LIN {X -0.095,Y -181.495,Z 926.751,A 0.000,B 0.000,C 90.000,E1 135.162} C_DIS
LIN {X 0.041,Y -187.011,Z 926.732,A 0.000,B 0.000,C 90.000,E1 131.757} C_DIS
LIN {X 0.043,Y -190.129,Z 926.723,A 0.000,B 0.000,C 90.000,E1 130.092} C_DIS
LIN {X -0.054,Y -193.964,Z 926.710,A 0.000,B 0.000,C 90.000,E1 127.890} C_DIS
LIN {X -0.123,Y -295.836,Z 926.710,A 0.000,B 0.000,C 90.000,E1 127.890} C_DIS
LIN {X 0.171,Y -297.593,Z 926.710,A 0.000,B 0.000,C 90.000,E1 127.810} C_DIS
LIN {X -0.111,Y -302.346,Z 926.709,A 0.000,B 0.000,C 90.000,E1 127.649} C_DIS
LIN {X -0.085,Y -305.517,Z 926.707,A 0.000,B 0.000,C 90.000,E1 127.363} C_DIS
LIN {X 0.048,Y -309.189,Z 926.705,A 0.000,B 0.000,C 90.000,E1 126.824} C_DIS
LIN {X 0.011,Y -310.829,Z 926.703,A 0.000,B 0.000,C 90.000,E1 126.503} C_DIS
LIN {X 0.039,Y -312.116,Z 926.701,A 0.000,B 0.000,C 90.000,E1 126.171} C_DIS
LIN {X 0.060,Y -323.509,Z 926.681,A 0.000,B 0.000,C 90.000,E1 122.625} C_DIS
LIN {X -0.009,Y -334.188,Z 926.666,A 0.000,B 0.000,C 90.000,E1 119.795} C_DIS
LIN {X 0.021,Y -346.235,Z 926.650,A 0.000,B 0.000,C 90.000,E1 117.001} C_DIS
LIN {X 0.081,Y -359.760,Z 926.635,A 0.000,B 0.000,C 90.000,E1 114.259} C_DIS
LIN {X -0.012,Y -373.117,Z 926.622,A 0.000,B 0.000,C 90.000,E1 111.897} C_DIS
LIN {X -0.042,Y -387.831,Z 926.609,A 0.000,B 0.000,C 90.000,E1 109.577} C_DIS
LIN {X 0.170,Y -404.006,Z 926.596,A 0.000,B 0.000,C 90.000,E1 107.275} C_DIS
LIN {X 0.157,Y -421.757,Z 926.584,A 0.000,B 0.000,C 90.000,E1 105.064} C_DIS
LIN {X -0.008,Y -441.147,Z 926.572,A 0.000,B 0.000,C 90.000,E1 102.939} C_DIS
LIN {X -0.050,Y -461.367,Z 926.561,A 0.000,B 0.000,C 90.000,E1 100.950} C_DIS
LIN {X -0.142,Y -466.507,Z 926.558,A 0.000,B 0.000,C 90.000,E1 100.489} C_DIS
LIN {X -0.104,Y -468.718,Z 926.557,A 0.000,B 0.000,C 90.000,E1 100.254} C_DIS
LIN {X -0.067,Y -470.389,Z 926.556,A 0.000,B 0.000,C 90.000,E1 100.018} C_DIS
LIN {X 0.249,Y -471.785,Z 926.554,A 0.000,B 0.000,C 90.000,E1 99.726} C_DIS
LIN {X 0.021,Y -472.823,Z 926.553,A 0.000,B 0.000,C 90.000,E1 99.500} C_DIS
LIN {X 0.205,Y -474.025,Z 926.550,A 0.000,B 0.000,C 90.000,E1 98.973} C_DIS
LIN {X -0.148,Y -474.224,Z 926.547,A 0.000,B 0.000,C 90.000,E1 98.511} C_DIS
LIN {X -0.023,Y -473.458,Z 926.544,A 0.000,B 0.000,C 90.000,E1 97.992} C_DIS
LIN {X 0.104,Y -471.602,Z 926.542,A 0.000,B 0.000,C 90.000,E1 97.473} C_DIS
LIN {X -0.181,Y -468.512,Z 926.539,A 0.000,B 0.000,C 90.000,E1 97.004} C_DIS
LIN {X 0.092,Y -452.500,Z 926.525,A 0.000,B 0.000,C 90.000,E1 94.416} C_DIS
LIN {X 0.019,Y -443.003,Z 926.516,A 0.000,B 0.000,C 90.000,E1 92.865} C_DIS
LIN {X 0.196,Y -433.326,Z 926.507,A 0.000,B 0.000,C 90.000,E1 91.260} C_DIS
LIN {X 0.126,Y -418.840,Z 926.494,A 0.000,B 0.000,C 90.000,E1 88.854} C_DIS
LIN {X -0.035,Y -407.917,Z 926.483,A 0.000,B 0.000,C 90.000,E1 86.963} C_DIS
LIN {X 0.066,Y -395.372,Z 926.471,A 0.000,B 0.000,C 90.000,E1 84.723} C_DIS
LIN {X -0.085,Y -384.384,Z 926.460,A 0.000,B 0.000,C 90.000,E1 82.761} C_DIS
LIN {X -0.038,Y -374.849,Z 926.450,A 0.000,B 0.000,C 90.000,E1 81.027} C_DIS
LIN {X -0.110,Y -365.068,Z 926.440,A 0.000,B 0.000,C 90.000,E1 79.285} C_DIS
LIN {X 0.090,Y -353.365,Z 926.429,A 0.000,B 0.000,C 90.000,E1 77.173} C_DIS
LIN {X 0.115,Y -341.692,Z 926.417,A 0.000,B 0.000,C 90.000,E1 75.046} C_DIS
LIN {X 0.018,Y -322.845,Z 926.396,A 0.000,B 0.000,C 90.000,E1 71.329} C_DIS
LIN {X 0.021,Y -310.954,Z 926.382,A 0.000,B 0.000,C 90.000,E1 68.773} C_DIS
LIN {X 0.064,Y -300.551,Z 926.369,A 0.000,B 0.000,C 90.000,E1 66.485} C_DIS
LIN {X -0.141,Y -291.623,Z 926.358,A 0.000,B 0.000,C 90.000,E1 64.537} C_DIS
LIN {X 0.004,Y -282.685,Z 926.347,A 0.000,B 0.000,C 90.000,E1 62.487} C_DIS
LIN {X 0.042,Y -272.142,Z 926.334,A 0.000,B 0.000,C 90.000,E1 60.078} C_DIS
LIN {X -0.056,Y -260.381,Z 926.318,A 0.000,B 0.000,C 90.000,E1 57.296} C_DIS
LIN {X -0.064,Y -248.093,Z 926.300,A 0.000,B 0.000,C 90.000,E1 54.069} C_DIS
LIN {X 0.105,Y -237.172,Z 926.282,A 0.000,B 0.000,C 90.000,E1 50.723} C_DIS
LIN {X -0.082,Y -227.137,Z 926.263,A 0.000,B 0.000,C 90.000,E1 47.391} C_DIS
LIN {X -0.137,Y -218.924,Z 926.246,A 0.000,B 0.000,C 90.000,E1 44.352} C_DIS
LIN {X -0.075,Y -211.261,Z 926.229,A 0.000,B 0.000,C 90.000,E1 41.229} C_DIS
LIN {X 0.000,Y -204.280,Z 926.211,A 0.000,B 0.000,C 90.000,E1 38.051} C_DIS
LIN {X -0.010,Y -196.202,Z 926.189,A 0.000,B 0.000,C 90.000,E1 34.040} C_DIS
LIN {X -0.076,Y -190.298,Z 926.171,A 0.000,B 0.000,C 90.000,E1 30.797} C_DIS
LIN {X 0.020,Y -185.028,Z 926.153,A 0.000,B 0.000,C 90.000,E1 27.462} C_DIS
LIN {X -0.024,Y -180.372,Z 926.134,A 0.000,B 0.000,C 90.000,E1 24.131} C_DIS
LIN {X 0.021,Y -176.434,Z 926.115,A 0.000,B 0.000,C 90.000,E1 20.737} C_DIS
LIN {X -0.059,Y -172.457,Z 926.092,A 0.000,B 0.000,C 90.000,E1 16.496} C_DIS
LIN {X -0.007,Y -169.607,Z 926.068,A 0.000,B 0.000,C 90.000,E1 12.175} C_DIS
LIN {X 0.048,Y -167.410,Z 926.034,A 0.000,B 0.000,C 90.000,E1 6.087} C_DIS
LIN {X 0.008,Y -168.434,Z 925.973,A 0.000,B 0.000,C 90.000,E1 355.179} C_DIS
LIN {X 0.001,Y -171.200,Z 925.944,A 0.000,B 0.000,C 90.000,E1 349.982} C_DIS
LIN {X -0.066,Y -174.623,Z 925.920,A 0.000,B 0.000,C 90.000,E1 345.700} C_DIS
LIN {X 0.076,Y -178.081,Z 925.901,A 0.000,B 0.000,C 90.000,E1 342.236} C_DIS
LIN {X -0.002,Y -183.377,Z 925.878,A 0.000,B 0.000,C 90.000,E1 338.028} C_DIS
LIN {X 0.049,Y -188.469,Z 925.859,A 0.000,B 0.000,C 90.000,E1 334.665} C_DIS
LIN {X -0.048,Y -194.337,Z 925.841,A 0.000,B 0.000,C 90.000,E1 331.385} C_DIS
LIN {X -0.057,Y -200.894,Z 925.823,A 0.000,B 0.000,C 90.000,E1 328.122} C_DIS
LIN {X -0.025,Y -207.916,Z 925.805,A 0.000,B 0.000,C 90.000,E1 324.895} C_DIS
LIN {X -0.012,Y -216.445,Z 925.785,A 0.000,B 0.000,C 90.000,E1 321.331} C_DIS
LIN {X -0.005,Y -225.714,Z 925.766,A 0.000,B 0.000,C 90.000,E1 317.838} C_DIS
LIN {X -0.012,Y -234.984,Z 925.749,A 0.000,B 0.000,C 90.000,E1 314.798} C_DIS
LIN {X -0.116,Y -245.275,Z 925.732,A 0.000,B 0.000,C 90.000,E1 311.838} C_DIS
LIN {X -0.111,Y -255.319,Z 925.718,A 0.000,B 0.000,C 90.000,E1 309.277} C_DIS
LIN {X 0.064,Y -268.084,Z 925.702,A 0.000,B 0.000,C 90.000,E1 306.377} C_DIS
LIN {X 0.157,Y -280.556,Z 925.689,A 0.000,B 0.000,C 90.000,E1 303.913} C_DIS
LIN {X 0.057,Y -298.031,Z 925.672,A 0.000,B 0.000,C 90.000,E1 300.875} C_DIS
LIN {X 0.103,Y -314.949,Z 925.657,A 0.000,B 0.000,C 90.000,E1 298.231} C_DIS
LIN {X 0.089,Y -328.966,Z 925.646,A 0.000,B 0.000,C 90.000,E1 296.309} C_DIS
LIN {X -0.077,Y -351.659,Z 925.631,A 0.000,B 0.000,C 90.000,E1 293.567} C_DIS
LIN {X 0.112,Y -369.983,Z 925.620,A 0.000,B 0.000,C 90.000,E1 291.535} C_DIS
LIN {X 0.017,Y -385.864,Z 925.610,A 0.000,B 0.000,C 90.000,E1 289.885} C_DIS
LIN {X -0.139,Y -401.502,Z 925.602,A 0.000,B 0.000,C 90.000,E1 288.290} C_DIS
LIN {X 0.173,Y -414.172,Z 925.594,A 0.000,B 0.000,C 90.000,E1 286.913} C_DIS
LIN {X 0.039,Y -424.176,Z 925.588,A 0.000,B 0.000,C 90.000,E1 285.843} C_DIS
LIN {X 0.220,Y -431.309,Z 925.584,A 0.000,B 0.000,C 90.000,E1 285.009} C_DIS
LIN {X -0.004,Y -442.623,Z 925.576,A 0.000,B 0.000,C 90.000,E1 283.703} C_DIS
LIN {X 0.024,Y -451.189,Z 925.570,A 0.000,B 0.000,C 90.000,E1 282.647} C_DIS
LIN {X -0.110,Y -461.234,Z 925.563,A 0.000,B 0.000,C 90.000,E1 281.366} C_DIS
LIN {X 0.142,Y -468.714,Z 925.557,A 0.000,B 0.000,C 90.000,E1 280.310} C_DIS
LIN {X 0.071,Y -474.002,Z 925.553,A 0.000,B 0.000,C 90.000,E1 279.557} C_DIS
LIN {X 0.053,Y -478.719,Z 925.549,A 0.000,B 0.000,C 90.000,E1 278.803} C_DIS
LIN {X 0.072,Y -482.786,Z 925.545,A 0.000,B 0.000,C 90.000,E1 278.049} C_DIS
LIN {X -0.236,Y -485.091,Z 925.542,A 0.000,B 0.000,C 90.000,E1 277.587} C_DIS
LIN {X -0.049,Y -487.043,Z 925.539,A 0.000,B 0.000,C 90.000,E1 277.068} C_DIS
LIN {X 0.148,Y -488.694,Z 925.536,A 0.000,B 0.000,C 90.000,E1 276.549} C_DIS
LIN {X -0.131,Y -490.011,Z 925.534,A 0.000,B 0.000,C 90.000,E1 276.087} C_DIS
LIN {X 0.086,Y -490.984,Z 925.531,A 0.000,B 0.000,C 90.000,E1 275.568} C_DIS
LIN {X -0.179,Y -491.590,Z 925.528,A 0.000,B 0.000,C 90.000,E1 275.106} C_DIS
LIN {X 0.049,Y -491.776,Z 925.526,A 0.000,B 0.000,C 90.000,E1 274.588} C_DIS
LIN {X -0.248,Y -491.574,Z 925.523,A 0.000,B 0.000,C 90.000,E1 274.131} C_DIS
LIN {X -0.017,Y -490.851,Z 925.520,A 0.000,B 0.000,C 90.000,E1 273.612} C_DIS
LIN {X 0.208,Y -489.636,Z 925.517,A 0.000,B 0.000,C 90.000,E1 273.094} C_DIS
LIN {X -0.086,Y -487.839,Z 925.515,A 0.000,B 0.000,C 90.000,E1 272.636} C_DIS
LIN {X 0.103,Y -485.340,Z 925.512,A 0.000,B 0.000,C 90.000,E1 272.121} C_DIS
LIN {X -0.192,Y -482.109,Z 925.509,A 0.000,B 0.000,C 90.000,E1 271.661} C_DIS
LIN {X -0.037,Y -477.985,Z 925.506,A 0.000,B 0.000,C 90.000,E1 271.146} C_DIS
LIN {X 0.097,Y -472.901,Z 925.504,A 0.000,B 0.000,C 90.000,E1 270.630} C_DIS
LIN {X -0.052,Y -467.036,Z 925.501,A 0.000,B 0.000,C 90.000,E1 270.172} C_DIS
LIN {X -0.218,Y -460.853,Z 925.499,A 0.000,B 0.000,C 90.000,E1 269.771} C_DIS
LIN {X 0.061,Y -454.296,Z 925.497,A 0.000,B 0.000,C 90.000,E1 269.370} C_DIS
LIN {X -0.181,Y -447.561,Z 925.495,A 0.000,B 0.000,C 90.000,E1 269.083} C_DIS
LIN {X -0.110,Y -440.479,Z 925.493,A 0.000,B 0.000,C 90.000,E1 268.797} C_DIS
LIN {X -0.106,Y -433.533,Z 925.492,A 0.000,B 0.000,C 90.000,E1 268.568} C_DIS
LIN {X 0.157,Y -426.244,Z 925.491,A 0.000,B 0.000,C 90.000,E1 268.339} C_DIS
LIN {X -0.164,Y -416.975,Z 925.490,A 0.000,B 0.000,C 90.000,E1 268.224} C_DIS
LIN {X 0.042,Y -406.402,Z 925.490,A 0.000,B 0.000,C 90.000,E1 268.108} C_DIS
LIN {X -0.008,Y -403.442,Z 925.490,A 0.000,B 0.000,C 90.000,E1 268.108} C_DIS
LIN {X -0.027,Y -181.141,Z 925.489,A 0.000,B 0.000,C 90.000,E1 268.108} C_DIS
LIN {X -0.037,Y -180.899,Z 925.474,A 0.000,B 0.000,C 90.000,E1 265.241} C_DIS
LIN {X -0.088,Y -180.212,Z 925.464,A 0.000,B 0.000,C 90.000,E1 263.571} C_DIS
LIN {X 0.042,Y -179.032,Z 925.445,A 0.000,B 0.000,C 90.000,E1 260.151} C_DIS
LIN {X -0.072,Y -178.687,Z 925.441,A 0.000,B 0.000,C 90.000,E1 259.342} C_DIS
LIN {X 0.040,Y -175.737,Z 925.412,A 0.000,B 0.000,C 90.000,E1 254.212} C_DIS
LIN {X 0.035,Y -171.921,Z 925.384,A 0.000,B 0.000,C 90.000,E1 249.082} C_DIS
LIN {X 0.010,Y -171.292,Z 925.379,A 0.000,B 0.000,C 90.000,E1 248.230} C_DIS
LIN {X 0.055,Y -167.557,Z 925.355,A 0.000,B 0.000,C 90.000,E1 243.896} C_DIS
LIN {X 0.068,Y -166.179,Z 925.345,A 0.000,B 0.000,C 90.000,E1 242.153} C_DIS
LIN {X 0.059,Y -162.950,Z 925.326,A 0.000,B 0.000,C 90.000,E1 238.663} C_DIS
LIN {X 0.106,Y -160.858,Z 925.311,A 0.000,B 0.000,C 90.000,E1 236.008} C_DIS
LIN {X 0.083,Y -157.634,Z 925.292,A 0.000,B 0.000,C 90.000,E1 232.477} C_DIS
LIN {X 0.021,Y -155.670,Z 925.277,A 0.000,B 0.000,C 90.000,E1 229.828} C_DIS
LIN {X 0.073,Y -151.938,Z 925.252,A 0.000,B 0.000,C 90.000,E1 225.324} C_DIS
LIN {X 0.088,Y -150.175,Z 925.237,A 0.000,B 0.000,C 90.000,E1 222.609} C_DIS
LIN {X 0.007,Y -146.951,Z 925.212,A 0.000,B 0.000,C 90.000,E1 218.096} C_DIS
LIN {X -0.004,Y -145.539,Z 925.196,A 0.000,B 0.000,C 90.000,E1 215.358} C_DIS
LIN {X 0.034,Y -142.935,Z 925.171,A 0.000,B 0.000,C 90.000,E1 210.747} C_DIS
LIN {X -0.031,Y -141.559,Z 925.150,A 0.000,B 0.000,C 90.000,E1 207.078} C_DIS
LIN {X 0.022,Y -139.408,Z 925.114,A 0.000,B 0.000,C 90.000,E1 200.556} C_DIS
LIN {X -0.057,Y -139.129,Z 925.104,A 0.000,B 0.000,C 90.000,E1 198.725} C_DIS
LIN {X -0.030,Y -138.351,Z 925.057,A 0.000,B 0.000,C 90.000,E1 190.310} C_DIS
LIN {X -0.042,Y -139.498,Z 925.005,A 0.000,B 0.000,C 90.000,E1 180.974} C_DIS
LIN {X 0.039,Y -141.121,Z 924.974,A 0.000,B 0.000,C 90.000,E1 175.355} C_DIS
LIN {X -0.008,Y -142.501,Z 924.959,A 0.000,B 0.000,C 90.000,E1 172.591} C_DIS
LIN {X -0.061,Y -144.757,Z 924.933,A 0.000,B 0.000,C 90.000,E1 167.993} C_DIS
LIN {X 0.029,Y -147.367,Z 924.913,A 0.000,B 0.000,C 90.000,E1 164.283} C_DIS
LIN {X -0.048,Y -150.695,Z 924.887,A 0.000,B 0.000,C 90.000,E1 159.752} C_DIS
LIN {X 0.035,Y -154.175,Z 924.867,A 0.000,B 0.000,C 90.000,E1 156.102} C_DIS
LIN {X -0.035,Y -157.609,Z 924.847,A 0.000,B 0.000,C 90.000,E1 152.538} C_DIS
LIN {X 0.053,Y -161.863,Z 924.828,A 0.000,B 0.000,C 90.000,E1 148.948} C_DIS
LIN {X -0.068,Y -166.053,Z 924.808,A 0.000,B 0.000,C 90.000,E1 145.468} C_DIS
LIN {X -0.077,Y -171.058,Z 924.789,A 0.000,B 0.000,C 90.000,E1 141.984} C_DIS
LIN {X -0.048,Y -175.929,Z 924.770,A 0.000,B 0.000,C 90.000,E1 138.528} C_DIS
LIN {X -0.055,Y -180.169,Z 924.755,A 0.000,B 0.000,C 90.000,E1 135.972} C_DIS
LIN {X -0.087,Y -185.586,Z 924.737,A 0.000,B 0.000,C 90.000,E1 132.609} C_DIS
LIN {X -0.038,Y -190.176,Z 924.723,A 0.000,B 0.000,C 90.000,E1 130.092} C_DIS
LIN {X 0.025,Y -193.923,Z 924.711,A 0.000,B 0.000,C 90.000,E1 127.890} C_DIS
LIN {X -0.014,Y -295.957,Z 924.711,A 0.000,B 0.000,C 90.000,E1 127.890} C_DIS
LIN {X 0.085,Y -300.709,Z 924.710,A 0.000,B 0.000,C 90.000,E1 127.729} C_DIS
LIN {X 0.003,Y -302.892,Z 924.709,A 0.000,B 0.000,C 90.000,E1 127.604} C_DIS
LIN {X -0.137,Y -306.757,Z 924.707,A 0.000,B 0.000,C 90.000,E1 127.237} C_DIS
LIN {X -0.134,Y -310.233,Z 924.704,A 0.000,B 0.000,C 90.000,E1 126.664} C_DIS
LIN {X 0.081,Y -311.626,Z 924.702,A 0.000,B 0.000,C 90.000,E1 126.297} C_DIS
LIN {X 0.039,Y -318.727,Z 924.689,A 0.000,B 0.000,C 90.000,E1 124.040} C_DIS
LIN {X 0.001,Y -328.768,Z 924.673,A 0.000,B 0.000,C 90.000,E1 121.180} C_DIS
LIN {X 0.028,Y -340.133,Z 924.658,A 0.000,B 0.000,C 90.000,E1 118.359} C_DIS
LIN {X 0.073,Y -352.917,Z 924.642,A 0.000,B 0.000,C 90.000,E1 115.591} C_DIS
LIN {X -0.042,Y -365.568,Z 924.629,A 0.000,B 0.000,C 90.000,E1 113.206} C_DIS
LIN {X 0.009,Y -379.521,Z 924.616,A 0.000,B 0.000,C 90.000,E1 110.844} C_DIS
LIN {X 0.006,Y -394.876,Z 924.603,A 0.000,B 0.000,C 90.000,E1 108.544} C_DIS
LIN {X -0.117,Y -411.743,Z 924.591,A 0.000,B 0.000,C 90.000,E1 106.315} C_DIS
LIN {X -0.064,Y -430.244,Z 924.578,A 0.000,B 0.000,C 90.000,E1 104.120} C_DIS
LIN {X 0.128,Y -450.112,Z 924.567,A 0.000,B 0.000,C 90.000,E1 102.007} C_DIS
LIN {X 0.198,Y -467.878,Z 924.557,A 0.000,B 0.000,C 90.000,E1 100.310} C_DIS
LIN {X 0.158,Y -469.812,Z 924.556,A 0.000,B 0.000,C 90.000,E1 100.074} C_DIS
LIN {X 0.037,Y -471.282,Z 924.555,A 0.000,B 0.000,C 90.000,E1 99.849} C_DIS
LIN {X 0.211,Y -473.299,Z 924.552,A 0.000,B 0.000,C 90.000,E1 99.321} C_DIS
LIN {X -0.151,Y -474.183,Z 924.549,A 0.000,B 0.000,C 90.000,E1 98.859} C_DIS
LIN {X -0.031,Y -474.091,Z 924.546,A 0.000,B 0.000,C 90.000,E1 98.341} C_DIS
LIN {X 0.161,Y -473.014,Z 924.544,A 0.000,B 0.000,C 90.000,E1 97.814} C_DIS
LIN {X -0.042,Y -472.058,Z 924.542,A 0.000,B 0.000,C 90.000,E1 97.587} C_DIS
LIN {X -0.182,Y -470.765,Z 924.541,A 0.000,B 0.000,C 90.000,E1 97.352} C_DIS
LIN {X -0.039,Y -453.129,Z 924.525,A 0.000,B 0.000,C 90.000,E1 94.531} C_DIS
LIN {X -0.099,Y -443.699,Z 924.516,A 0.000,B 0.000,C 90.000,E1 92.980} C_DIS
LIN {X -0.182,Y -432.428,Z 924.506,A 0.000,B 0.000,C 90.000,E1 91.146} C_DIS
LIN {X -0.153,Y -416.397,Z 924.491,A 0.000,B 0.000,C 90.000,E1 88.453} C_DIS
LIN {X 0.063,Y -405.418,Z 924.481,A 0.000,B 0.000,C 90.000,E1 86.502} C_DIS
LIN {X 0.088,Y -394.435,Z 924.470,A 0.000,B 0.000,C 90.000,E1 84.546} C_DIS
LIN {X -0.123,Y -383.435,Z 924.459,A 0.000,B 0.000,C 90.000,E1 82.591} C_DIS
LIN {X -0.038,Y -373.879,Z 924.449,A 0.000,B 0.000,C 90.000,E1 80.849} C_DIS
LIN {X -0.104,Y -365.737,Z 924.441,A 0.000,B 0.000,C 90.000,E1 79.398} C_DIS
LIN {X 0.080,Y -355.726,Z 924.431,A 0.000,B 0.000,C 90.000,E1 77.589} C_DIS
LIN {X 0.151,Y -343.999,Z 924.419,A 0.000,B 0.000,C 90.000,E1 75.463} C_DIS
LIN {X 0.032,Y -324.991,Z 924.399,A 0.000,B 0.000,C 90.000,E1 71.764} C_DIS
LIN {X 0.080,Y -313.063,Z 924.385,A 0.000,B 0.000,C 90.000,E1 69.209} C_DIS
LIN {X -0.115,Y -302.672,Z 924.372,A 0.000,B 0.000,C 90.000,E1 66.975} C_DIS
LIN {X -0.005,Y -293.773,Z 924.361,A 0.000,B 0.000,C 90.000,E1 64.973} C_DIS
LIN {X 0.050,Y -284.841,Z 924.350,A 0.000,B 0.000,C 90.000,E1 62.948} C_DIS
LIN {X -0.108,Y -274.283,Z 924.336,A 0.000,B 0.000,C 90.000,E1 60.589} C_DIS
LIN {X 0.027,Y -263.917,Z 924.323,A 0.000,B 0.000,C 90.000,E1 58.122} C_DIS
LIN {X 0.108,Y -251.273,Z 924.305,A 0.000,B 0.000,C 90.000,E1 54.895} C_DIS
LIN {X 0.078,Y -241.239,Z 924.289,A 0.000,B 0.000,C 90.000,E1 51.984} C_DIS
LIN {X 0.021,Y -230.929,Z 924.270,A 0.000,B 0.000,C 90.000,E1 48.647} C_DIS
LIN {X -0.110,Y -222.470,Z 924.253,A 0.000,B 0.000,C 90.000,E1 45.648} C_DIS
LIN {X 0.029,Y -214.580,Z 924.236,A 0.000,B 0.000,C 90.000,E1 42.528} C_DIS
LIN {X -0.008,Y -207.346,Z 924.219,A 0.000,B 0.000,C 90.000,E1 39.402} C_DIS
LIN {X -0.004,Y -200.701,Z 924.201,A 0.000,B 0.000,C 90.000,E1 36.217} C_DIS
LIN {X 0.088,Y -194.418,Z 924.183,A 0.000,B 0.000,C 90.000,E1 32.959} C_DIS
LIN {X -0.023,Y -188.726,Z 924.165,A 0.000,B 0.000,C 90.000,E1 29.716} C_DIS
LIN {X -0.061,Y -183.643,Z 924.147,A 0.000,B 0.000,C 90.000,E1 26.411} C_DIS
LIN {X 0.037,Y -179.251,Z 924.128,A 0.000,B 0.000,C 90.000,E1 23.025} C_DIS
LIN {X 0.056,Y -175.510,Z 924.109,A 0.000,B 0.000,C 90.000,E1 19.631} C_DIS
LIN {X 0.008,Y -171.847,Z 924.085,A 0.000,B 0.000,C 90.000,E1 15.371} C_DIS
LIN {X 0.002,Y -168.879,Z 924.057,A 0.000,B 0.000,C 90.000,E1 10.197} C_DIS
LIN {X -0.005,Y -169.464,Z 923.964,A 0.000,B 0.000,C 90.000,E1 353.451} C_DIS
LIN {X 0.060,Y -172.087,Z 923.940,A 0.000,B 0.000,C 90.000,E1 349.106} C_DIS
LIN {X 0.062,Y -175.694,Z 923.916,A 0.000,B 0.000,C 90.000,E1 344.810} C_DIS
LIN {X 0.060,Y -179.312,Z 923.897,A 0.000,B 0.000,C 90.000,E1 341.402} C_DIS
LIN {X 0.041,Y -183.617,Z 923.878,A 0.000,B 0.000,C 90.000,E1 338.028} C_DIS
LIN {X -0.071,Y -188.722,Z 923.859,A 0.000,B 0.000,C 90.000,E1 334.717} C_DIS
LIN {X 0.010,Y -194.621,Z 923.841,A 0.000,B 0.000,C 90.000,E1 331.385} C_DIS
LIN {X 0.010,Y -201.196,Z 923.823,A 0.000,B 0.000,C 90.000,E1 328.122} C_DIS
LIN {X 0.052,Y -208.184,Z 923.805,A 0.000,B 0.000,C 90.000,E1 324.895} C_DIS
LIN {X 0.001,Y -215.746,Z 923.787,A 0.000,B 0.000,C 90.000,E1 321.743} C_DIS
LIN {X 0.017,Y -224.902,Z 923.768,A 0.000,B 0.000,C 90.000,E1 318.243} C_DIS
LIN {X -0.013,Y -234.042,Z 923.751,A 0.000,B 0.000,C 90.000,E1 315.202} C_DIS
LIN {X 0.023,Y -244.181,Z 923.734,A 0.000,B 0.000,C 90.000,E1 312.204} C_DIS
LIN {X 0.023,Y -255.543,Z 923.718,A 0.000,B 0.000,C 90.000,E1 309.277} C_DIS
LIN {X -0.006,Y -268.251,Z 923.702,A 0.000,B 0.000,C 90.000,E1 306.423} C_DIS
LIN {X -0.076,Y -280.639,Z 923.689,A 0.000,B 0.000,C 90.000,E1 303.992} C_DIS
LIN {X -0.031,Y -298.021,Z 923.672,A 0.000,B 0.000,C 90.000,E1 300.924} C_DIS
LIN {X 0.001,Y -314.874,Z 923.657,A 0.000,B 0.000,C 90.000,E1 298.281} C_DIS
LIN {X -0.023,Y -328.780,Z 923.646,A 0.000,B 0.000,C 90.000,E1 296.360} C_DIS
LIN {X 0.026,Y -351.472,Z 923.631,A 0.000,B 0.000,C 90.000,E1 293.567} C_DIS
LIN {X -0.085,Y -372.537,Z 923.618,A 0.000,B 0.000,C 90.000,E1 291.280} C_DIS
LIN {X -0.112,Y -388.292,Z 923.609,A 0.000,B 0.000,C 90.000,E1 289.631} C_DIS
LIN {X 0.228,Y -401.332,Z 923.602,A 0.000,B 0.000,C 90.000,E1 288.236} C_DIS
LIN {X 0.168,Y -413.952,Z 923.594,A 0.000,B 0.000,C 90.000,E1 286.913} C_DIS
LIN {X 0.046,Y -423.968,Z 923.588,A 0.000,B 0.000,C 90.000,E1 285.843} C_DIS
LIN {X -0.161,Y -431.098,Z 923.584,A 0.000,B 0.000,C 90.000,E1 285.064} C_DIS
LIN {X 0.031,Y -442.469,Z 923.576,A 0.000,B 0.000,C 90.000,E1 283.703} C_DIS
LIN {X 0.057,Y -451.015,Z 923.570,A 0.000,B 0.000,C 90.000,E1 282.647} C_DIS
LIN {X -0.079,Y -461.081,Z 923.563,A 0.000,B 0.000,C 90.000,E1 281.366} C_DIS
LIN {X 0.171,Y -468.575,Z 923.557,A 0.000,B 0.000,C 90.000,E1 280.310} C_DIS
LIN {X 0.100,Y -473.867,Z 923.553,A 0.000,B 0.000,C 90.000,E1 279.557} C_DIS
LIN {X 0.082,Y -478.673,Z 923.549,A 0.000,B 0.000,C 90.000,E1 278.803} C_DIS
LIN {X 0.100,Y -482.766,Z 923.545,A 0.000,B 0.000,C 90.000,E1 278.049} C_DIS
LIN {X -0.208,Y -485.077,Z 923.542,A 0.000,B 0.000,C 90.000,E1 277.587} C_DIS
LIN {X -0.021,Y -487.051,Z 923.539,A 0.000,B 0.000,C 90.000,E1 277.068} C_DIS
LIN {X 0.176,Y -488.706,Z 923.536,A 0.000,B 0.000,C 90.000,E1 276.549} C_DIS
LIN {X -0.103,Y -490.052,Z 923.534,A 0.000,B 0.000,C 90.000,E1 276.087} C_DIS
LIN {X 0.115,Y -491.018,Z 923.531,A 0.000,B 0.000,C 90.000,E1 275.568} C_DIS
LIN {X -0.150,Y -491.632,Z 923.528,A 0.000,B 0.000,C 90.000,E1 275.106} C_DIS
LIN {X 0.077,Y -491.863,Z 923.526,A 0.000,B 0.000,C 90.000,E1 274.588} C_DIS
LIN {X -0.219,Y -491.638,Z 923.523,A 0.000,B 0.000,C 90.000,E1 274.131} C_DIS
LIN {X 0.012,Y -490.934,Z 923.520,A 0.000,B 0.000,C 90.000,E1 273.612} C_DIS
LIN {X 0.237,Y -489.765,Z 923.517,A 0.000,B 0.000,C 90.000,E1 273.094} C_DIS
LIN {X -0.056,Y -487.969,Z 923.515,A 0.000,B 0.000,C 90.000,E1 272.636} C_DIS
LIN {X 0.133,Y -485.501,Z 923.512,A 0.000,B 0.000,C 90.000,E1 272.121} C_DIS
LIN {X -0.022,Y -484.041,Z 923.510,A 0.000,B 0.000,C 90.000,E1 271.892} C_DIS
LIN {X 0.158,Y -480.403,Z 923.508,A 0.000,B 0.000,C 90.000,E1 271.375} C_DIS
LIN {X -0.174,Y -475.858,Z 923.505,A 0.000,B 0.000,C 90.000,E1 270.917} C_DIS
LIN {X 0.072,Y -470.456,Z 923.502,A 0.000,B 0.000,C 90.000,E1 270.401} C_DIS
LIN {X 0.149,Y -464.526,Z 923.500,A 0.000,B 0.000,C 90.000,E1 269.943} C_DIS
LIN {X 0.161,Y -458.177,Z 923.498,A 0.000,B 0.000,C 90.000,E1 269.542} C_DIS
LIN {X 0.146,Y -451.496,Z 923.496,A 0.000,B 0.000,C 90.000,E1 269.198} C_DIS
LIN {X 0.055,Y -444.732,Z 923.494,A 0.000,B 0.000,C 90.000,E1 268.912} C_DIS
LIN {X -0.142,Y -437.810,Z 923.493,A 0.000,B 0.000,C 90.000,E1 268.682} C_DIS
LIN {X -0.026,Y -430.706,Z 923.491,A 0.000,B 0.000,C 90.000,E1 268.453} C_DIS
LIN {X -0.077,Y -422.903,Z 923.490,A 0.000,B 0.000,C 90.000,E1 268.282} C_DIS
LIN {X -0.140,Y -413.957,Z 923.490,A 0.000,B 0.000,C 90.000,E1 268.165} C_DIS
LIN {X -0.116,Y -405.152,Z 923.489,A 0.000,B 0.000,C 90.000,E1 268.108} C_DIS
LIN {X -0.076,Y -181.138,Z 923.489,A 0.000,B 0.000,C 90.000,E1 268.108} C_DIS
LIN {X -0.090,Y -180.897,Z 923.473,A 0.000,B 0.000,C 90.000,E1 265.241} C_DIS
LIN {X -0.067,Y -179.844,Z 923.459,A 0.000,B 0.000,C 90.000,E1 262.704} C_DIS
LIN {X -0.009,Y -179.028,Z 923.445,A 0.000,B 0.000,C 90.000,E1 260.151} C_DIS
LIN {X 0.053,Y -178.676,Z 923.441,A 0.000,B 0.000,C 90.000,E1 259.285} C_DIS
LIN {X -0.011,Y -175.726,Z 923.412,A 0.000,B 0.000,C 90.000,E1 254.212} C_DIS
LIN {X 0.005,Y -172.443,Z 923.389,A 0.000,B 0.000,C 90.000,E1 249.934} C_DIS
LIN {X -0.040,Y -171.276,Z 923.379,A 0.000,B 0.000,C 90.000,E1 248.230} C_DIS
LIN {X 0.006,Y -167.544,Z 923.355,A 0.000,B 0.000,C 90.000,E1 243.896} C_DIS
LIN {X 0.020,Y -166.162,Z 923.345,A 0.000,B 0.000,C 90.000,E1 242.153} C_DIS
LIN {X 0.010,Y -162.937,Z 923.326,A 0.000,B 0.000,C 90.000,E1 238.663} C_DIS
LIN {X -0.012,Y -161.607,Z 923.316,A 0.000,B 0.000,C 90.000,E1 236.914} C_DIS
LIN {X -0.037,Y -159.133,Z 923.301,A 0.000,B 0.000,C 90.000,E1 234.276} C_DIS
LIN {X -0.027,Y -155.655,Z 923.277,A 0.000,B 0.000,C 90.000,E1 229.828} C_DIS
LIN {X 0.026,Y -151.925,Z 923.252,A 0.000,B 0.000,C 90.000,E1 225.324} C_DIS
LIN {X 0.041,Y -150.161,Z 923.237,A 0.000,B 0.000,C 90.000,E1 222.609} C_DIS
LIN {X -0.038,Y -146.941,Z 923.212,A 0.000,B 0.000,C 90.000,E1 218.096} C_DIS
LIN {X 0.069,Y -145.528,Z 923.196,A 0.000,B 0.000,C 90.000,E1 215.311} C_DIS
LIN {X -0.011,Y -142.927,Z 923.171,A 0.000,B 0.000,C 90.000,E1 210.747} C_DIS
LIN {X -0.011,Y -141.550,Z 923.150,A 0.000,B 0.000,C 90.000,E1 207.052} C_DIS
LIN {X -0.023,Y -139.405,Z 923.114,A 0.000,B 0.000,C 90.000,E1 200.556} C_DIS
LIN {X 0.032,Y -139.123,Z 923.104,A 0.000,B 0.000,C 90.000,E1 198.671} C_DIS
LIN {X 0.063,Y -138.351,Z 923.057,A 0.000,B 0.000,C 90.000,E1 190.254} C_DIS
LIN {X 0.053,Y -139.502,Z 923.005,A 0.000,B 0.000,C 90.000,E1 180.917} C_DIS
LIN {X -0.006,Y -141.129,Z 922.974,A 0.000,B 0.000,C 90.000,E1 175.355} C_DIS
LIN {X -0.053,Y -142.510,Z 922.959,A 0.000,B 0.000,C 90.000,E1 172.591} C_DIS
LIN {X 0.035,Y -144.768,Z 922.933,A 0.000,B 0.000,C 90.000,E1 167.937} C_DIS
LIN {X -0.016,Y -147.381,Z 922.913,A 0.000,B 0.000,C 90.000,E1 164.283} C_DIS
LIN {X 0.047,Y -150.710,Z 922.887,A 0.000,B 0.000,C 90.000,E1 159.699} C_DIS
LIN {X -0.013,Y -154.191,Z 922.867,A 0.000,B 0.000,C 90.000,E1 156.102} C_DIS
LIN {X 0.057,Y -157.628,Z 922.847,A 0.000,B 0.000,C 90.000,E1 152.487} C_DIS
LIN {X 0.005,Y -161.885,Z 922.828,A 0.000,B 0.000,C 90.000,E1 148.948} C_DIS
LIN {X -0.023,Y -166.074,Z 922.808,A 0.000,B 0.000,C 90.000,E1 145.435} C_DIS
LIN {X -0.022,Y -171.082,Z 922.789,A 0.000,B 0.000,C 90.000,E1 141.949} C_DIS
LIN {X 0.033,Y -175.955,Z 922.769,A 0.000,B 0.000,C 90.000,E1 138.485} C_DIS
LIN {X -0.107,Y -180.198,Z 922.755,A 0.000,B 0.000,C 90.000,E1 135.972} C_DIS
LIN {X 0.122,Y -185.614,Z 922.736,A 0.000,B 0.000,C 90.000,E1 132.528} C_DIS
LIN {X -0.091,Y -190.209,Z 922.723,A 0.000,B 0.000,C 90.000,E1 130.092} C_DIS
LIN {X 0.078,Y -193.895,Z 922.711,A 0.000,B 0.000,C 90.000,E1 127.890} C_DIS
LIN {X 0.067,Y -296.537,Z 922.711,A 0.000,B 0.000,C 90.000,E1 127.890} C_DIS
LIN {X -0.093,Y -298.037,Z 922.710,A 0.000,B 0.000,C 90.000,E1 127.890} C_DIS
LIN {X -0.083,Y -303.289,Z 922.709,A 0.000,B 0.000,C 90.000,E1 127.604} C_DIS
LIN {X 0.097,Y -306.505,Z 922.707,A 0.000,B 0.000,C 90.000,E1 127.237} C_DIS
LIN {X 0.056,Y -310.084,Z 922.704,A 0.000,B 0.000,C 90.000,E1 126.664} C_DIS
LIN {X -0.163,Y -311.491,Z 922.702,A 0.000,B 0.000,C 90.000,E1 126.377} C_DIS
LIN {X 0.129,Y -315.528,Z 922.695,A 0.000,B 0.000,C 90.000,E1 125.025} C_DIS
LIN {X -0.177,Y -326.281,Z 922.677,A 0.000,B 0.000,C 90.000,E1 121.878} C_DIS
LIN {X -0.052,Y -337.327,Z 922.661,A 0.000,B 0.000,C 90.000,E1 119.027} C_DIS
LIN {X 0.076,Y -349.769,Z 922.646,A 0.000,B 0.000,C 90.000,E1 116.232} C_DIS
LIN {X 0.089,Y -363.721,Z 922.631,A 0.000,B 0.000,C 90.000,E1 113.515} C_DIS
LIN {X 0.098,Y -377.490,Z 922.618,A 0.000,B 0.000,C 90.000,E1 111.153} C_DIS
LIN {X 0.049,Y -392.644,Z 922.605,A 0.000,B 0.000,C 90.000,E1 108.852} C_DIS
LIN {X -0.122,Y -409.295,Z 922.592,A 0.000,B 0.000,C 90.000,E1 106.622} C_DIS
LIN {X -0.015,Y -427.563,Z 922.580,A 0.000,B 0.000,C 90.000,E1 104.411} C_DIS
LIN {X 0.005,Y -447.315,Z 922.568,A 0.000,B 0.000,C 90.000,E1 102.299} C_DIS
LIN {X -0.065,Y -467.625,Z 922.558,A 0.000,B 0.000,C 90.000,E1 100.366} C_DIS
LIN {X -0.169,Y -469.604,Z 922.556,A 0.000,B 0.000,C 90.000,E1 100.141} C_DIS
LIN {X -0.189,Y -471.109,Z 922.555,A 0.000,B 0.000,C 90.000,E1 99.905} C_DIS
LIN {X 0.130,Y -472.321,Z 922.553,A 0.000,B 0.000,C 90.000,E1 99.613} C_DIS
LIN {X -0.018,Y -473.207,Z 922.552,A 0.000,B 0.000,C 90.000,E1 99.378} C_DIS
LIN {X 0.093,Y -474.154,Z 922.549,A 0.000,B 0.000,C 90.000,E1 98.859} C_DIS
LIN {X -0.256,Y -474.124,Z 922.547,A 0.000,B 0.000,C 90.000,E1 98.398} C_DIS
LIN {X -0.065,Y -473.113,Z 922.544,A 0.000,B 0.000,C 90.000,E1 97.871} C_DIS
LIN {X 0.200,Y -472.196,Z 922.542,A 0.000,B 0.000,C 90.000,E1 97.587} C_DIS
LIN {X 0.059,Y -470.951,Z 922.541,A 0.000,B 0.000,C 90.000,E1 97.352} C_DIS
LIN {X 0.200,Y -453.345,Z 922.525,A 0.000,B 0.000,C 90.000,E1 94.531} C_DIS
LIN {X 0.139,Y -443.949,Z 922.517,A 0.000,B 0.000,C 90.000,E1 92.980} C_DIS
LIN {X -0.106,Y -434.329,Z 922.508,A 0.000,B 0.000,C 90.000,E1 91.432} C_DIS
LIN {X -0.135,Y -419.804,Z 922.495,A 0.000,B 0.000,C 90.000,E1 89.026} C_DIS
LIN {X 0.134,Y -408.819,Z 922.484,A 0.000,B 0.000,C 90.000,E1 87.078} C_DIS
LIN {X -0.141,Y -396.226,Z 922.471,A 0.000,B 0.000,C 90.000,E1 84.894} C_DIS
LIN {X 0.122,Y -385.224,Z 922.461,A 0.000,B 0.000,C 90.000,E1 82.875} C_DIS
LIN {X 0.183,Y -375.690,Z 922.451,A 0.000,B 0.000,C 90.000,E1 81.141} C_DIS
LIN {X 0.124,Y -365.999,Z 922.441,A 0.000,B 0.000,C 90.000,E1 79.398} C_DIS
LIN {X -0.041,Y -355.976,Z 922.431,A 0.000,B 0.000,C 90.000,E1 77.645} C_DIS
LIN {X 0.042,Y -344.257,Z 922.420,A 0.000,B 0.000,C 90.000,E1 75.519} C_DIS
LIN {X -0.017,Y -326.746,Z 922.401,A 0.000,B 0.000,C 90.000,E1 72.127} C_DIS
LIN {X 0.006,Y -313.305,Z 922.385,A 0.000,B 0.000,C 90.000,E1 69.263} C_DIS
LIN {X 0.101,Y -302.913,Z 922.372,A 0.000,B 0.000,C 90.000,E1 66.975} C_DIS
LIN {X -0.057,Y -294.036,Z 922.361,A 0.000,B 0.000,C 90.000,E1 65.025} C_DIS
LIN {X 0.010,Y -285.100,Z 922.350,A 0.000,B 0.000,C 90.000,E1 62.999} C_DIS
LIN {X 0.102,Y -274.548,Z 922.337,A 0.000,B 0.000,C 90.000,E1 60.589} C_DIS
LIN {X -0.129,Y -264.187,Z 922.323,A 0.000,B 0.000,C 90.000,E1 58.201} C_DIS
LIN {X -0.037,Y -251.500,Z 922.305,A 0.000,B 0.000,C 90.000,E1 54.975} C_DIS
LIN {X -0.058,Y -241.458,Z 922.289,A 0.000,B 0.000,C 90.000,E1 52.065} C_DIS
LIN {X 0.049,Y -231.196,Z 922.271,A 0.000,B 0.000,C 90.000,E1 48.690} C_DIS
LIN {X 0.090,Y -222.757,Z 922.254,A 0.000,B 0.000,C 90.000,E1 45.648} C_DIS
LIN {X -0.074,Y -214.888,Z 922.237,A 0.000,B 0.000,C 90.000,E1 42.609} C_DIS
LIN {X 0.061,Y -207.635,Z 922.219,A 0.000,B 0.000,C 90.000,E1 39.439} C_DIS
LIN {X -0.002,Y -199.404,Z 922.197,A 0.000,B 0.000,C 90.000,E1 35.471} C_DIS
LIN {X 0.062,Y -193.243,Z 922.179,A 0.000,B 0.000,C 90.000,E1 32.212} C_DIS
LIN {X -0.009,Y -187.703,Z 922.161,A 0.000,B 0.000,C 90.000,E1 28.949} C_DIS
LIN {X 0.096,Y -182.773,Z 922.142,A 0.000,B 0.000,C 90.000,E1 25.591} C_DIS
LIN {X -0.063,Y -178.551,Z 922.124,A 0.000,B 0.000,C 90.000,E1 22.280} C_DIS
LIN {X 0.040,Y -174.173,Z 922.100,A 0.000,B 0.000,C 90.000,E1 18.000} C_DIS
LIN {X 0.026,Y -170.964,Z 922.076,A 0.000,B 0.000,C 90.000,E1 13.716} C_DIS
LIN {X -0.079,Y -168.486,Z 922.047,A 0.000,B 0.000,C 90.000,E1 8.568} C_DIS
LIN {X 0.006,Y -169.330,Z 921.968,A 0.000,B 0.000,C 90.000,E1 354.318} C_DIS
LIN {X 0.037,Y -171.735,Z 921.944,A 0.000,B 0.000,C 90.000,E1 349.982} C_DIS
LIN {X -0.014,Y -175.155,Z 921.921,A 0.000,B 0.000,C 90.000,E1 345.700} C_DIS
LIN {X -0.075,Y -179.562,Z 921.897,A 0.000,B 0.000,C 90.000,E1 341.456} C_DIS
LIN {X 0.014,Y -183.860,Z 921.878,A 0.000,B 0.000,C 90.000,E1 338.050} C_DIS
LIN {X -0.022,Y -188.972,Z 921.859,A 0.000,B 0.000,C 90.000,E1 334.717} C_DIS
LIN {X 0.068,Y -194.917,Z 921.841,A 0.000,B 0.000,C 90.000,E1 331.385} C_DIS
LIN {X 0.078,Y -201.494,Z 921.823,A 0.000,B 0.000,C 90.000,E1 328.122} C_DIS
LIN {X 0.129,Y -208.458,Z 921.805,A 0.000,B 0.000,C 90.000,E1 324.895} C_DIS
LIN {X 0.088,Y -216.036,Z 921.788,A 0.000,B 0.000,C 90.000,E1 321.743} C_DIS
LIN {X 0.115,Y -225.182,Z 921.768,A 0.000,B 0.000,C 90.000,E1 318.243} C_DIS
LIN {X -0.070,Y -234.307,Z 921.751,A 0.000,B 0.000,C 90.000,E1 315.243} C_DIS
LIN {X -0.020,Y -244.431,Z 921.735,A 0.000,B 0.000,C 90.000,E1 312.243} C_DIS
LIN {X -0.042,Y -255.763,Z 921.718,A 0.000,B 0.000,C 90.000,E1 309.322} C_DIS
LIN {X -0.020,Y -268.415,Z 921.703,A 0.000,B 0.000,C 90.000,E1 306.457} C_DIS
LIN {X 0.079,Y -280.727,Z 921.689,A 0.000,B 0.000,C 90.000,E1 303.992} C_DIS
LIN {X 0.136,Y -298.029,Z 921.672,A 0.000,B 0.000,C 90.000,E1 300.924} C_DIS
LIN {X 0.029,Y -314.785,Z 921.657,A 0.000,B 0.000,C 90.000,E1 298.309} C_DIS
LIN {X 0.158,Y -328.585,Z 921.647,A 0.000,B 0.000,C 90.000,E1 296.360} C_DIS
LIN {X -0.062,Y -353.593,Z 921.630,A 0.000,B 0.000,C 90.000,E1 293.334} C_DIS
LIN {X 0.086,Y -374.390,Z 921.617,A 0.000,B 0.000,C 90.000,E1 291.046} C_DIS
LIN {X 0.041,Y -390.137,Z 921.608,A 0.000,B 0.000,C 90.000,E1 289.396} C_DIS
LIN {X 0.026,Y -403.161,Z 921.600,A 0.000,B 0.000,C 90.000,E1 288.055} C_DIS
LIN {X -0.118,Y -415.826,Z 921.593,A 0.000,B 0.000,C 90.000,E1 286.732} C_DIS
LIN {X -0.102,Y -425.592,Z 921.587,A 0.000,B 0.000,C 90.000,E1 285.662} C_DIS
LIN {X -0.135,Y -434.984,Z 921.581,A 0.000,B 0.000,C 90.000,E1 284.592} C_DIS
LIN {X -0.201,Y -443.975,Z 921.575,A 0.000,B 0.000,C 90.000,E1 283.536} C_DIS
LIN {X -0.155,Y -452.455,Z 921.569,A 0.000,B 0.000,C 90.000,E1 282.479} C_DIS
LIN {X -0.006,Y -460.483,Z 921.563,A 0.000,B 0.000,C 90.000,E1 281.422} C_DIS
LIN {X 0.237,Y -468.020,Z 921.558,A 0.000,B 0.000,C 90.000,E1 280.366} C_DIS
LIN {X 0.018,Y -475.047,Z 921.552,A 0.000,B 0.000,C 90.000,E1 279.378} C_DIS
LIN {X 0.001,Y -479.720,Z 921.548,A 0.000,B 0.000,C 90.000,E1 278.624} C_DIS
LIN {X 0.029,Y -483.670,Z 921.544,A 0.000,B 0.000,C 90.000,E1 277.871} C_DIS
LIN {X 0.026,Y -486.826,Z 921.540,A 0.000,B 0.000,C 90.000,E1 277.125} C_DIS
LIN {X -0.259,Y -488.519,Z 921.537,A 0.000,B 0.000,C 90.000,E1 276.663} C_DIS
LIN {X -0.054,Y -489.915,Z 921.534,A 0.000,B 0.000,C 90.000,E1 276.144} C_DIS
LIN {X 0.162,Y -490.946,Z 921.531,A 0.000,B 0.000,C 90.000,E1 275.625} C_DIS
LIN {X -0.104,Y -491.612,Z 921.529,A 0.000,B 0.000,C 90.000,E1 275.163} C_DIS
LIN {X 0.123,Y -491.893,Z 921.526,A 0.000,B 0.000,C 90.000,E1 274.645} C_DIS
LIN {X -0.174,Y -491.748,Z 921.523,A 0.000,B 0.000,C 90.000,E1 274.188} C_DIS
LIN {X 0.058,Y -491.143,Z 921.520,A 0.000,B 0.000,C 90.000,E1 273.669} C_DIS
LIN {X -0.233,Y -490.051,Z 921.518,A 0.000,B 0.000,C 90.000,E1 273.212} C_DIS
LIN {X -0.010,Y -488.336,Z 921.515,A 0.000,B 0.000,C 90.000,E1 272.694} C_DIS
LIN {X -0.159,Y -487.279,Z 921.514,A 0.000,B 0.000,C 90.000,E1 272.465} C_DIS
LIN {X 0.027,Y -484.590,Z 921.511,A 0.000,B 0.000,C 90.000,E1 271.949} C_DIS
LIN {X 0.209,Y -481.120,Z 921.508,A 0.000,B 0.000,C 90.000,E1 271.432} C_DIS
LIN {X 0.048,Y -479.069,Z 921.507,A 0.000,B 0.000,C 90.000,E1 271.203} C_DIS
LIN {X 0.187,Y -474.189,Z 921.504,A 0.000,B 0.000,C 90.000,E1 270.688} C_DIS
LIN {X -0.069,Y -468.402,Z 921.501,A 0.000,B 0.000,C 90.000,E1 270.229} C_DIS
LIN {X 0.148,Y -462.349,Z 921.499,A 0.000,B 0.000,C 90.000,E1 269.771} C_DIS
LIN {X -0.153,Y -455.808,Z 921.497,A 0.000,B 0.000,C 90.000,E1 269.427} C_DIS
LIN {X -0.019,Y -449.132,Z 921.495,A 0.000,B 0.000,C 90.000,E1 269.083} C_DIS
LIN {X 0.017,Y -442.319,Z 921.493,A 0.000,B 0.000,C 90.000,E1 268.797} C_DIS
LIN {X -0.074,Y -435.280,Z 921.492,A 0.000,B 0.000,C 90.000,E1 268.568} C_DIS
LIN {X 0.117,Y -427.931,Z 921.491,A 0.000,B 0.000,C 90.000,E1 268.339} C_DIS
LIN {X 0.175,Y -419.511,Z 921.490,A 0.000,B 0.000,C 90.000,E1 268.167} C_DIS
LIN {X -0.010,Y -411.653,Z 921.490,A 0.000,B 0.000,C 90.000,E1 268.108} C_DIS
LIN {X 0.140,Y -404.770,Z 921.489,A 0.000,B 0.000,C 90.000,E1 268.051} C_DIS
LIN {X 0.038,Y -181.135,Z 921.489,A 0.000,B 0.000,C 90.000,E1 268.051} C_DIS
LIN {X 0.059,Y -180.907,Z 921.475,A 0.000,B 0.000,C 90.000,E1 265.469} C_DIS
LIN {X -0.064,Y -180.745,Z 921.470,A 0.000,B 0.000,C 90.000,E1 264.666} C_DIS
LIN {X 0.005,Y -178.836,Z 921.442,A 0.000,B 0.000,C 90.000,E1 259.577} C_DIS
LIN {X -0.098,Y -175.880,Z 921.414,A 0.000,B 0.000,C 90.000,E1 254.519} C_DIS
LIN {X 0.008,Y -174.542,Z 921.404,A 0.000,B 0.000,C 90.000,E1 252.779} C_DIS
LIN {X 0.100,Y -171.526,Z 921.381,A 0.000,B 0.000,C 90.000,E1 248.465} C_DIS
LIN {X 0.086,Y -167.752,Z 921.357,A 0.000,B 0.000,C 90.000,E1 244.152} C_DIS
LIN {X 0.025,Y -166.456,Z 921.347,A 0.000,B 0.000,C 90.000,E1 242.436} C_DIS
LIN {X 0.014,Y -163.172,Z 921.328,A 0.000,B 0.000,C 90.000,E1 238.948} C_DIS
LIN {X 0.063,Y -161.131,Z 921.313,A 0.000,B 0.000,C 90.000,E1 236.294} C_DIS
LIN {X -0.034,Y -157.152,Z 921.288,A 0.000,B 0.000,C 90.000,E1 231.904} C_DIS
LIN {X -0.011,Y -155.885,Z 921.278,A 0.000,B 0.000,C 90.000,E1 230.114} C_DIS
LIN {X -0.053,Y -152.135,Z 921.253,A 0.000,B 0.000,C 90.000,E1 225.648} C_DIS
LIN {X -0.032,Y -150.384,Z 921.238,A 0.000,B 0.000,C 90.000,E1 222.933} C_DIS
LIN {X -0.008,Y -147.117,Z 921.213,A 0.000,B 0.000,C 90.000,E1 218.382} C_DIS
LIN {X -0.017,Y -145.681,Z 921.198,A 0.000,B 0.000,C 90.000,E1 215.644} C_DIS
LIN {X -0.019,Y -143.064,Z 921.172,A 0.000,B 0.000,C 90.000,E1 211.052} C_DIS
LIN {X 0.038,Y -141.686,Z 921.152,A 0.000,B 0.000,C 90.000,E1 207.334} C_DIS
LIN {X 0.016,Y -139.459,Z 921.116,A 0.000,B 0.000,C 90.000,E1 200.844} C_DIS
LIN {X 0.067,Y -139.193,Z 921.105,A 0.000,B 0.000,C 90.000,E1 198.960} C_DIS
LIN {X -0.046,Y -138.324,Z 921.054,A 0.000,B 0.000,C 90.000,E1 189.670} C_DIS
LIN {X -0.041,Y -139.453,Z 921.007,A 0.000,B 0.000,C 90.000,E1 181.260} C_DIS
LIN {X 0.039,Y -141.000,Z 920.976,A 0.000,B 0.000,C 90.000,E1 175.641} C_DIS
LIN {X -0.011,Y -142.755,Z 920.955,A 0.000,B 0.000,C 90.000,E1 171.951} C_DIS
LIN {X -0.056,Y -145.157,Z 920.930,A 0.000,B 0.000,C 90.000,E1 167.353} C_DIS
LIN {X -0.063,Y -147.780,Z 920.909,A 0.000,B 0.000,C 90.000,E1 163.685} C_DIS
LIN {X 0.017,Y -150.458,Z 920.889,A 0.000,B 0.000,C 90.000,E1 160.007} C_DIS
LIN {X -0.050,Y -153.907,Z 920.869,A 0.000,B 0.000,C 90.000,E1 156.410} C_DIS
LIN {X 0.015,Y -157.317,Z 920.849,A 0.000,B 0.000,C 90.000,E1 152.794} C_DIS
LIN {X -0.039,Y -161.506,Z 920.829,A 0.000,B 0.000,C 90.000,E1 149.253} C_DIS
LIN {X -0.023,Y -165.705,Z 920.810,A 0.000,B 0.000,C 90.000,E1 145.722} C_DIS
LIN {X 0.103,Y -170.650,Z 920.790,A 0.000,B 0.000,C 90.000,E1 142.190} C_DIS
LIN {X 0.017,Y -175.525,Z 920.771,A 0.000,B 0.000,C 90.000,E1 138.771} C_DIS
LIN {X 0.010,Y -181.145,Z 920.752,A 0.000,B 0.000,C 90.000,E1 135.364} C_DIS
LIN {X 0.008,Y -186.598,Z 920.733,A 0.000,B 0.000,C 90.000,E1 132.000} C_DIS
LIN {X 0.078,Y -191.207,Z 920.719,A 0.000,B 0.000,C 90.000,E1 129.483} C_DIS
LIN {X 0.014,Y -193.849,Z 920.711,A 0.000,B 0.000,C 90.000,E1 127.935} C_DIS
LIN {X -0.012,Y -295.428,Z 920.711,A 0.000,B 0.000,C 90.000,E1 127.935} C_DIS
LIN {X 0.008,Y -299.078,Z 920.710,A 0.000,B 0.000,C 90.000,E1 127.855} C_DIS
LIN {X 0.046,Y -302.111,Z 920.709,A 0.000,B 0.000,C 90.000,E1 127.684} C_DIS
LIN {X -0.011,Y -305.727,Z 920.708,A 0.000,B 0.000,C 90.000,E1 127.363} C_DIS
LIN {X 0.043,Y -309.305,Z 920.705,A 0.000,B 0.000,C 90.000,E1 126.824} C_DIS
LIN {X 0.006,Y -310.864,Z 920.703,A 0.000,B 0.000,C 90.000,E1 126.503} C_DIS
LIN {X 0.035,Y -312.088,Z 920.701,A 0.000,B 0.000,C 90.000,E1 126.171} C_DIS
LIN {X 0.055,Y -323.449,Z 920.681,A 0.000,B 0.000,C 90.000,E1 122.625} C_DIS
LIN {X -0.017,Y -334.128,Z 920.666,A 0.000,B 0.000,C 90.000,E1 119.795} C_DIS
LIN {X 0.012,Y -346.175,Z 920.650,A 0.000,B 0.000,C 90.000,E1 117.001} C_DIS
LIN {X 0.069,Y -359.700,Z 920.635,A 0.000,B 0.000,C 90.000,E1 114.259} C_DIS
LIN {X -0.026,Y -373.058,Z 920.622,A 0.000,B 0.000,C 90.000,E1 111.897} C_DIS
LIN {X -0.059,Y -387.772,Z 920.609,A 0.000,B 0.000,C 90.000,E1 109.577} C_DIS
LIN {X 0.153,Y -403.947,Z 920.596,A 0.000,B 0.000,C 90.000,E1 107.275} C_DIS
LIN {X 0.137,Y -421.700,Z 920.584,A 0.000,B 0.000,C 90.000,E1 105.064} C_DIS
LIN {X -0.031,Y -441.091,Z 920.572,A 0.000,B 0.000,C 90.000,E1 102.939} C_DIS
LIN {X -0.075,Y -461.311,Z 920.561,A 0.000,B 0.000,C 90.000,E1 100.950} C_DIS
LIN {X -0.166,Y -466.452,Z 920.558,A 0.000,B 0.000,C 90.000,E1 100.489} C_DIS
LIN {X -0.129,Y -468.677,Z 920.557,A 0.000,B 0.000,C 90.000,E1 100.254} C_DIS
LIN {X -0.092,Y -470.358,Z 920.556,A 0.000,B 0.000,C 90.000,E1 100.018} C_DIS
LIN {X 0.223,Y -471.762,Z 920.554,A 0.000,B 0.000,C 90.000,E1 99.726} C_DIS
LIN {X -0.005,Y -472.806,Z 920.553,A 0.000,B 0.000,C 90.000,E1 99.500} C_DIS
LIN {X 0.179,Y -474.019,Z 920.550,A 0.000,B 0.000,C 90.000,E1 98.973} C_DIS
LIN {X -0.174,Y -474.230,Z 920.547,A 0.000,B 0.000,C 90.000,E1 98.511} C_DIS
LIN {X -0.049,Y -473.473,Z 920.544,A 0.000,B 0.000,C 90.000,E1 97.992} C_DIS
LIN {X 0.078,Y -471.631,Z 920.542,A 0.000,B 0.000,C 90.000,E1 97.473} C_DIS
LIN {X -0.206,Y -468.536,Z 920.539,A 0.000,B 0.000,C 90.000,E1 97.004} C_DIS
LIN {X -0.171,Y -451.034,Z 920.523,A 0.000,B 0.000,C 90.000,E1 94.188} C_DIS
LIN {X -0.002,Y -443.191,Z 920.516,A 0.000,B 0.000,C 90.000,E1 92.865} C_DIS
LIN {X 0.179,Y -433.578,Z 920.507,A 0.000,B 0.000,C 90.000,E1 91.260} C_DIS
LIN {X 0.115,Y -419.086,Z 920.494,A 0.000,B 0.000,C 90.000,E1 88.854} C_DIS
LIN {X -0.041,Y -408.075,Z 920.483,A 0.000,B 0.000,C 90.000,E1 86.963} C_DIS
LIN {X 0.064,Y -395.479,Z 920.471,A 0.000,B 0.000,C 90.000,E1 84.723} C_DIS
LIN {X -0.045,Y -382.894,Z 920.458,A 0.000,B 0.000,C 90.000,E1 82.470} C_DIS
LIN {X -0.024,Y -373.321,Z 920.448,A 0.000,B 0.000,C 90.000,E1 80.735} C_DIS
LIN {X -0.107,Y -365.207,Z 920.440,A 0.000,B 0.000,C 90.000,E1 79.285} C_DIS
LIN {X 0.095,Y -353.508,Z 920.429,A 0.000,B 0.000,C 90.000,E1 77.173} C_DIS
LIN {X 0.036,Y -340.180,Z 920.415,A 0.000,B 0.000,C 90.000,E1 74.755} C_DIS
LIN {X 0.031,Y -323.012,Z 920.396,A 0.000,B 0.000,C 90.000,E1 71.329} C_DIS
LIN {X 0.116,Y -312.616,Z 920.384,A 0.000,B 0.000,C 90.000,E1 69.082} C_DIS
LIN {X -0.092,Y -302.246,Z 920.371,A 0.000,B 0.000,C 90.000,E1 66.847} C_DIS
LIN {X 0.011,Y -293.374,Z 920.360,A 0.000,B 0.000,C 90.000,E1 64.845} C_DIS
LIN {X 0.059,Y -284.419,Z 920.349,A 0.000,B 0.000,C 90.000,E1 62.820} C_DIS
LIN {X -0.105,Y -273.891,Z 920.336,A 0.000,B 0.000,C 90.000,E1 60.461} C_DIS
LIN {X 0.015,Y -263.540,Z 920.322,A 0.000,B 0.000,C 90.000,E1 57.995} C_DIS
LIN {X 0.086,Y -250.927,Z 920.304,A 0.000,B 0.000,C 90.000,E1 54.769} C_DIS
LIN {X -0.142,Y -242.172,Z 920.290,A 0.000,B 0.000,C 90.000,E1 52.271} C_DIS
LIN {X -0.008,Y -231.898,Z 920.272,A 0.000,B 0.000,C 90.000,E1 48.895} C_DIS
LIN {X -0.097,Y -223.430,Z 920.255,A 0.000,B 0.000,C 90.000,E1 45.891} C_DIS
LIN {X 0.067,Y -215.559,Z 920.238,A 0.000,B 0.000,C 90.000,E1 42.771} C_DIS
LIN {X 0.055,Y -208.228,Z 920.220,A 0.000,B 0.000,C 90.000,E1 39.644} C_DIS
LIN {X -0.077,Y -201.624,Z 920.203,A 0.000,B 0.000,C 90.000,E1 36.503} C_DIS
LIN {X 0.042,Y -195.334,Z 920.185,A 0.000,B 0.000,C 90.000,E1 33.245} C_DIS
LIN {X -0.041,Y -189.583,Z 920.167,A 0.000,B 0.000,C 90.000,E1 30.001} C_DIS
LIN {X 0.033,Y -184.459,Z 920.148,A 0.000,B 0.000,C 90.000,E1 26.668} C_DIS
LIN {X -0.017,Y -180.036,Z 920.130,A 0.000,B 0.000,C 90.000,E1 23.334} C_DIS
LIN {X 0.023,Y -176.240,Z 920.111,A 0.000,B 0.000,C 90.000,E1 19.939} C_DIS
LIN {X 0.048,Y -172.512,Z 920.087,A 0.000,B 0.000,C 90.000,E1 15.662} C_DIS
LIN {X 0.063,Y -169.490,Z 920.058,A 0.000,B 0.000,C 90.000,E1 10.489} C_DIS
LIN {X -0.022,Y -167.832,Z 920.005,A 0.000,B 0.000,C 90.000,E1 0.974} C_DIS
LIN {X 0.016,Y -169.588,Z 919.968,A 0.000,B 0.000,C 90.000,E1 354.318} C_DIS
LIN {X -0.071,Y -172.599,Z 919.940,A 0.000,B 0.000,C 90.000,E1 349.162} C_DIS
LIN {X -0.052,Y -176.216,Z 919.916,A 0.000,B 0.000,C 90.000,E1 344.866} C_DIS
LIN {X -0.040,Y -179.817,Z 919.897,A 0.000,B 0.000,C 90.000,E1 341.456} C_DIS
LIN {X 0.056,Y -184.111,Z 919.878,A 0.000,B 0.000,C 90.000,E1 338.050} C_DIS
LIN {X 0.027,Y -189.239,Z 919.860,A 0.000,B 0.000,C 90.000,E1 334.717} C_DIS
LIN {X -0.046,Y -195.225,Z 919.841,A 0.000,B 0.000,C 90.000,E1 331.435} C_DIS
LIN {X 0.038,Y -201.782,Z 919.823,A 0.000,B 0.000,C 90.000,E1 328.152} C_DIS
LIN {X -0.084,Y -208.736,Z 919.805,A 0.000,B 0.000,C 90.000,E1 324.975} C_DIS
LIN {X 0.042,Y -216.326,Z 919.788,A 0.000,B 0.000,C 90.000,E1 321.778} C_DIS
LIN {X -0.034,Y -224.410,Z 919.770,A 0.000,B 0.000,C 90.000,E1 318.690} C_DIS
LIN {X -0.074,Y -233.361,Z 919.753,A 0.000,B 0.000,C 90.000,E1 315.648} C_DIS
LIN {X 0.115,Y -243.351,Z 919.737,A 0.000,B 0.000,C 90.000,E1 312.609} C_DIS
LIN {X -0.094,Y -254.526,Z 919.721,A 0.000,B 0.000,C 90.000,E1 309.725} C_DIS
LIN {X -0.152,Y -266.933,Z 919.705,A 0.000,B 0.000,C 90.000,E1 306.870} C_DIS
LIN {X -0.092,Y -279.002,Z 919.691,A 0.000,B 0.000,C 90.000,E1 304.405} C_DIS
LIN {X -0.103,Y -296.056,Z 919.674,A 0.000,B 0.000,C 90.000,E1 301.337} C_DIS
LIN {X -0.121,Y -312.510,Z 919.659,A 0.000,B 0.000,C 90.000,E1 298.693} C_DIS
LIN {X -0.043,Y -325.999,Z 919.649,A 0.000,B 0.000,C 90.000,E1 296.744} C_DIS
LIN {X -0.095,Y -350.915,Z 919.631,A 0.000,B 0.000,C 90.000,E1 293.643} C_DIS
LIN {X -0.104,Y -371.809,Z 919.618,A 0.000,B 0.000,C 90.000,E1 291.334} C_DIS
LIN {X -0.119,Y -384.984,Z 919.611,A 0.000,B 0.000,C 90.000,E1 289.939} C_DIS
LIN {X -0.102,Y -400.683,Z 919.602,A 0.000,B 0.000,C 90.000,E1 288.308} C_DIS
LIN {X 0.052,Y -410.793,Z 919.596,A 0.000,B 0.000,C 90.000,E1 287.221} C_DIS
LIN {X 0.084,Y -420.729,Z 919.590,A 0.000,B 0.000,C 90.000,E1 286.150} C_DIS
LIN {X 0.108,Y -430.490,Z 919.584,A 0.000,B 0.000,C 90.000,E1 285.064} C_DIS
LIN {X -0.238,Y -441.910,Z 919.576,A 0.000,B 0.000,C 90.000,E1 283.772} C_DIS
LIN {X -0.118,Y -450.540,Z 919.570,A 0.000,B 0.000,C 90.000,E1 282.703} C_DIS
LIN {X -0.091,Y -458.665,Z 919.565,A 0.000,B 0.000,C 90.000,E1 281.658} C_DIS
LIN {X 0.131,Y -466.313,Z 919.559,A 0.000,B 0.000,C 90.000,E1 280.602} C_DIS
LIN {X -0.105,Y -473.481,Z 919.553,A 0.000,B 0.000,C 90.000,E1 279.613} C_DIS
LIN {X -0.131,Y -478.365,Z 919.549,A 0.000,B 0.000,C 90.000,E1 278.859} C_DIS
LIN {X -0.118,Y -482.566,Z 919.545,A 0.000,B 0.000,C 90.000,E1 278.106} C_DIS
LIN {X 0.052,Y -484.958,Z 919.542,A 0.000,B 0.000,C 90.000,E1 277.587} C_DIS
LIN {X -0.244,Y -486.966,Z 919.539,A 0.000,B 0.000,C 90.000,E1 277.125} C_DIS
LIN {X -0.049,Y -488.657,Z 919.537,A 0.000,B 0.000,C 90.000,E1 276.606} C_DIS
LIN {X 0.159,Y -490.022,Z 919.534,A 0.000,B 0.000,C 90.000,E1 276.087} C_DIS
LIN {X -0.113,Y -491.038,Z 919.531,A 0.000,B 0.000,C 90.000,E1 275.625} C_DIS
LIN {X 0.111,Y -491.690,Z 919.528,A 0.000,B 0.000,C 90.000,E1 275.106} C_DIS
LIN {X -0.151,Y -491.966,Z 919.526,A 0.000,B 0.000,C 90.000,E1 274.645} C_DIS
LIN {X 0.043,Y -491.780,Z 919.523,A 0.000,B 0.000,C 90.000,E1 274.131} C_DIS
LIN {X -0.216,Y -491.155,Z 919.520,A 0.000,B 0.000,C 90.000,E1 273.669} C_DIS
LIN {X -0.017,Y -490.044,Z 919.518,A 0.000,B 0.000,C 90.000,E1 273.154} C_DIS
LIN {X 0.206,Y -488.345,Z 919.515,A 0.000,B 0.000,C 90.000,E1 272.636} C_DIS
LIN {X -0.089,Y -485.969,Z 919.512,A 0.000,B 0.000,C 90.000,E1 272.178} C_DIS
LIN {X 0.103,Y -482.909,Z 919.509,A 0.000,B 0.000,C 90.000,E1 271.661} C_DIS
LIN {X -0.218,Y -478.979,Z 919.507,A 0.000,B 0.000,C 90.000,E1 271.203} C_DIS
LIN {X -0.078,Y -474.099,Z 919.504,A 0.000,B 0.000,C 90.000,E1 270.688} C_DIS
LIN {X 0.186,Y -468.420,Z 919.501,A 0.000,B 0.000,C 90.000,E1 270.172} C_DIS
LIN {X -0.066,Y -462.341,Z 919.499,A 0.000,B 0.000,C 90.000,E1 269.771} C_DIS
LIN {X 0.097,Y -455.800,Z 919.497,A 0.000,B 0.000,C 90.000,E1 269.370} C_DIS
LIN {X -0.208,Y -449.213,Z 919.495,A 0.000,B 0.000,C 90.000,E1 269.083} C_DIS
LIN {X -0.164,Y -442.413,Z 919.493,A 0.000,B 0.000,C 90.000,E1 268.797} C_DIS
LIN {X 0.186,Y -435.387,Z 919.492,A 0.000,B 0.000,C 90.000,E1 268.511} C_DIS
LIN {X -0.043,Y -427.990,Z 919.491,A 0.000,B 0.000,C 90.000,E1 268.339} C_DIS
LIN {X 0.072,Y -419.914,Z 919.490,A 0.000,B 0.000,C 90.000,E1 268.165} C_DIS
LIN {X -0.118,Y -412.209,Z 919.489,A 0.000,B 0.000,C 90.000,E1 268.108} C_DIS
LIN {X -0.021,Y -404.409,Z 919.489,A 0.000,B 0.000,C 90.000,E1 268.051} C_DIS
LIN {X -0.035,Y -181.131,Z 919.489,A 0.000,B 0.000,C 90.000,E1 268.051} C_DIS
LIN {X 0.007,Y -180.907,Z 919.475,A 0.000,B 0.000,C 90.000,E1 265.469} C_DIS
LIN {X 0.063,Y -180.738,Z 919.470,A 0.000,B 0.000,C 90.000,E1 264.609} C_DIS
LIN {X -0.015,Y -178.827,Z 919.442,A 0.000,B 0.000,C 90.000,E1 259.567} C_DIS
LIN {X 0.066,Y -175.872,Z 919.414,A 0.000,B 0.000,C 90.000,E1 254.448} C_DIS
LIN {X -0.105,Y -173.844,Z 919.399,A 0.000,B 0.000,C 90.000,E1 251.945} C_DIS
LIN {X 0.050,Y -171.513,Z 919.380,A 0.000,B 0.000,C 90.000,E1 248.465} C_DIS
LIN {X 0.036,Y -167.740,Z 919.356,A 0.000,B 0.000,C 90.000,E1 244.152} C_DIS
LIN {X 0.052,Y -166.439,Z 919.347,A 0.000,B 0.000,C 90.000,E1 242.410} C_DIS
LIN {X -0.036,Y -163.157,Z 919.327,A 0.000,B 0.000,C 90.000,E1 238.948} C_DIS
LIN {X 0.014,Y -161.114,Z 919.313,A 0.000,B 0.000,C 90.000,E1 236.294} C_DIS
LIN {X -0.003,Y -157.839,Z 919.293,A 0.000,B 0.000,C 90.000,E1 232.763} C_DIS
LIN {X 0.061,Y -155.872,Z 919.278,A 0.000,B 0.000,C 90.000,E1 230.070} C_DIS
LIN {X 0.009,Y -152.122,Z 919.253,A 0.000,B 0.000,C 90.000,E1 225.607} C_DIS
LIN {X 0.024,Y -150.372,Z 919.238,A 0.000,B 0.000,C 90.000,E1 222.894} C_DIS
LIN {X -0.054,Y -147.106,Z 919.213,A 0.000,B 0.000,C 90.000,E1 218.382} C_DIS
LIN {X 0.056,Y -145.673,Z 919.198,A 0.000,B 0.000,C 90.000,E1 215.598} C_DIS
LIN {X 0.058,Y -143.056,Z 919.172,A 0.000,B 0.000,C 90.000,E1 211.003} C_DIS
LIN {X -0.007,Y -141.678,Z 919.152,A 0.000,B 0.000,C 90.000,E1 207.334} C_DIS
LIN {X -0.028,Y -139.455,Z 919.116,A 0.000,B 0.000,C 90.000,E1 200.844} C_DIS
LIN {X 0.023,Y -139.189,Z 919.105,A 0.000,B 0.000,C 90.000,E1 198.960} C_DIS
LIN {X 0.046,Y -138.323,Z 919.054,A 0.000,B 0.000,C 90.000,E1 189.613} C_DIS
LIN {X 0.053,Y -139.457,Z 919.007,A 0.000,B 0.000,C 90.000,E1 181.203} C_DIS
LIN {X -0.006,Y -141.008,Z 918.976,A 0.000,B 0.000,C 90.000,E1 175.641} C_DIS
LIN {X -0.057,Y -142.762,Z 918.955,A 0.000,B 0.000,C 90.000,E1 171.951} C_DIS
LIN {X 0.039,Y -145.168,Z 918.930,A 0.000,B 0.000,C 90.000,E1 167.297} C_DIS
LIN {X 0.032,Y -147.791,Z 918.909,A 0.000,B 0.000,C 90.000,E1 163.630} C_DIS
LIN {X -0.031,Y -150.473,Z 918.889,A 0.000,B 0.000,C 90.000,E1 160.007} C_DIS
LIN {X 0.043,Y -153.925,Z 918.869,A 0.000,B 0.000,C 90.000,E1 156.357} C_DIS
LIN {X -0.033,Y -157.336,Z 918.849,A 0.000,B 0.000,C 90.000,E1 152.794} C_DIS
LIN {X 0.051,Y -161.528,Z 918.829,A 0.000,B 0.000,C 90.000,E1 149.203} C_DIS
LIN {X 0.064,Y -165.727,Z 918.809,A 0.000,B 0.000,C 90.000,E1 145.674} C_DIS
LIN {X 0.051,Y -170.677,Z 918.790,A 0.000,B 0.000,C 90.000,E1 142.190} C_DIS
LIN {X -0.036,Y -175.551,Z 918.771,A 0.000,B 0.000,C 90.000,E1 138.771} C_DIS
LIN {X 0.084,Y -181.170,Z 918.752,A 0.000,B 0.000,C 90.000,E1 135.324} C_DIS
LIN {X -0.046,Y -186.626,Z 918.733,A 0.000,B 0.000,C 90.000,E1 132.000} C_DIS
LIN {X 0.024,Y -191.234,Z 918.719,A 0.000,B 0.000,C 90.000,E1 129.483} C_DIS
LIN {X -0.035,Y -193.812,Z 918.711,A 0.000,B 0.000,C 90.000,E1 127.971} C_DIS
LIN {X 0.093,Y -295.542,Z 918.711,A 0.000,B 0.000,C 90.000,E1 127.935} C_DIS
LIN {X 0.160,Y -299.873,Z 918.710,A 0.000,B 0.000,C 90.000,E1 127.810} C_DIS
LIN {X -0.058,Y -303.034,Z 918.709,A 0.000,B 0.000,C 90.000,E1 127.649} C_DIS
LIN {X 0.071,Y -306.704,Z 918.707,A 0.000,B 0.000,C 90.000,E1 127.237} C_DIS
LIN {X 0.027,Y -308.651,Z 918.705,A 0.000,B 0.000,C 90.000,E1 126.950} C_DIS
LIN {X -0.017,Y -310.185,Z 918.704,A 0.000,B 0.000,C 90.000,E1 126.664} C_DIS
LIN {X -0.046,Y -311.531,Z 918.702,A 0.000,B 0.000,C 90.000,E1 126.343} C_DIS
LIN {X 0.025,Y -324.003,Z 918.680,A 0.000,B 0.000,C 90.000,E1 122.467} C_DIS
LIN {X 0.082,Y -334.757,Z 918.665,A 0.000,B 0.000,C 90.000,E1 119.617} C_DIS
LIN {X -0.168,Y -346.884,Z 918.649,A 0.000,B 0.000,C 90.000,E1 116.873} C_DIS
LIN {X -0.097,Y -360.497,Z 918.634,A 0.000,B 0.000,C 90.000,E1 114.131} C_DIS
LIN {X 0.168,Y -373.938,Z 918.621,A 0.000,B 0.000,C 90.000,E1 111.716} C_DIS
LIN {X 0.167,Y -388.743,Z 918.608,A 0.000,B 0.000,C 90.000,E1 109.396} C_DIS
LIN {X 0.025,Y -405.016,Z 918.595,A 0.000,B 0.000,C 90.000,E1 107.149} C_DIS
LIN {X -0.085,Y -422.875,Z 918.583,A 0.000,B 0.000,C 90.000,E1 104.954} C_DIS
LIN {X -0.199,Y -442.347,Z 918.571,A 0.000,B 0.000,C 90.000,E1 102.827} C_DIS
LIN {X -0.157,Y -462.604,Z 918.560,A 0.000,B 0.000,C 90.000,E1 100.838} C_DIS
LIN {X -0.144,Y -467.668,Z 918.557,A 0.000,B 0.000,C 90.000,E1 100.366} C_DIS
LIN {X -0.250,Y -469.642,Z 918.556,A 0.000,B 0.000,C 90.000,E1 100.141} C_DIS
LIN {X 0.193,Y -471.142,Z 918.555,A 0.000,B 0.000,C 90.000,E1 99.849} C_DIS
LIN {X 0.048,Y -472.350,Z 918.553,A 0.000,B 0.000,C 90.000,E1 99.613} C_DIS
LIN {X -0.100,Y -473.232,Z 918.552,A 0.000,B 0.000,C 90.000,E1 99.378} C_DIS
LIN {X 0.011,Y -474.173,Z 918.549,A 0.000,B 0.000,C 90.000,E1 98.859} C_DIS
LIN {X 0.130,Y -474.136,Z 918.546,A 0.000,B 0.000,C 90.000,E1 98.341} C_DIS
LIN {X -0.146,Y -473.118,Z 918.544,A 0.000,B 0.000,C 90.000,E1 97.871} C_DIS
LIN {X 0.119,Y -472.198,Z 918.542,A 0.000,B 0.000,C 90.000,E1 97.587} C_DIS
LIN {X -0.022,Y -470.947,Z 918.541,A 0.000,B 0.000,C 90.000,E1 97.352} C_DIS
LIN {X -0.112,Y -451.801,Z 918.524,A 0.000,B 0.000,C 90.000,E1 94.302} C_DIS
LIN {X -0.190,Y -442.402,Z 918.515,A 0.000,B 0.000,C 90.000,E1 92.751} C_DIS
LIN {X -0.018,Y -432.782,Z 918.506,A 0.000,B 0.000,C 90.000,E1 91.146} C_DIS
LIN {X -0.095,Y -418.322,Z 918.493,A 0.000,B 0.000,C 90.000,E1 88.740} C_DIS
LIN {X 0.167,Y -407.295,Z 918.482,A 0.000,B 0.000,C 90.000,E1 86.788} C_DIS
LIN {X -0.172,Y -394.677,Z 918.470,A 0.000,B 0.000,C 90.000,E1 84.609} C_DIS
LIN {X 0.084,Y -382.079,Z 918.457,A 0.000,B 0.000,C 90.000,E1 82.299} C_DIS
LIN {X 0.083,Y -372.503,Z 918.448,A 0.000,B 0.000,C 90.000,E1 80.566} C_DIS
LIN {X 0.049,Y -364.372,Z 918.440,A 0.000,B 0.000,C 90.000,E1 79.106} C_DIS
LIN {X -0.111,Y -352.690,Z 918.428,A 0.000,B 0.000,C 90.000,E1 77.048} C_DIS
LIN {X 0.153,Y -339.386,Z 918.414,A 0.000,B 0.000,C 90.000,E1 74.574} C_DIS
LIN {X 0.119,Y -322.295,Z 918.395,A 0.000,B 0.000,C 90.000,E1 71.148} C_DIS
LIN {X -0.107,Y -311.898,Z 918.383,A 0.000,B 0.000,C 90.000,E1 68.954} C_DIS
LIN {X -0.043,Y -301.555,Z 918.370,A 0.000,B 0.000,C 90.000,E1 66.666} C_DIS
LIN {X 0.037,Y -291.216,Z 918.357,A 0.000,B 0.000,C 90.000,E1 64.332} C_DIS
LIN {X 0.041,Y -282.223,Z 918.346,A 0.000,B 0.000,C 90.000,E1 62.308} C_DIS
LIN {X 0.136,Y -270.246,Z 918.331,A 0.000,B 0.000,C 90.000,E1 59.537} C_DIS
LIN {X -0.111,Y -257.165,Z 918.313,A 0.000,B 0.000,C 90.000,E1 56.421} C_DIS
LIN {X -0.014,Y -249.050,Z 918.301,A 0.000,B 0.000,C 90.000,E1 54.242} C_DIS
LIN {X 0.047,Y -238.186,Z 918.283,A 0.000,B 0.000,C 90.000,E1 50.928} C_DIS
LIN {X -0.043,Y -229.332,Z 918.266,A 0.000,B 0.000,C 90.000,E1 47.957} C_DIS
LIN {X -0.049,Y -221.106,Z 918.249,A 0.000,B 0.000,C 90.000,E1 44.919} C_DIS
LIN {X -0.092,Y -213.331,Z 918.232,A 0.000,B 0.000,C 90.000,E1 41.838} C_DIS
LIN {X 0.003,Y -206.283,Z 918.215,A 0.000,B 0.000,C 90.000,E1 38.669} C_DIS
LIN {X 0.024,Y -199.821,Z 918.197,A 0.000,B 0.000,C 90.000,E1 35.471} C_DIS
LIN {X 0.099,Y -193.671,Z 918.179,A 0.000,B 0.000,C 90.000,E1 32.212} C_DIS
LIN {X 0.037,Y -188.139,Z 918.161,A 0.000,B 0.000,C 90.000,E1 28.949} C_DIS
LIN {X -0.013,Y -183.217,Z 918.142,A 0.000,B 0.000,C 90.000,E1 25.643} C_DIS
LIN {X 0.088,Y -178.045,Z 918.119,A 0.000,B 0.000,C 90.000,E1 21.408} C_DIS
LIN {X 0.057,Y -173.913,Z 918.095,A 0.000,B 0.000,C 90.000,E1 17.166} C_DIS
LIN {X 0.079,Y -170.483,Z 918.067,A 0.000,B 0.000,C 90.000,E1 12.007} C_DIS
LIN {X 0.029,Y -168.339,Z 918.033,A 0.000,B 0.000,C 90.000,E1 5.967} C_DIS
LIN {X 0.040,Y -169.485,Z 917.973,A 0.000,B 0.000,C 90.000,E1 355.179} C_DIS
LIN {X 0.072,Y -172.246,Z 917.944,A 0.000,B 0.000,C 90.000,E1 349.982} C_DIS
LIN {X 0.038,Y -175.674,Z 917.921,A 0.000,B 0.000,C 90.000,E1 345.700} C_DIS
LIN {X -0.006,Y -180.067,Z 917.897,A 0.000,B 0.000,C 90.000,E1 341.456} C_DIS
LIN {X -0.073,Y -184.359,Z 917.878,A 0.000,B 0.000,C 90.000,E1 338.103} C_DIS
LIN {X 0.076,Y -189.538,Z 917.860,A 0.000,B 0.000,C 90.000,E1 334.717} C_DIS
LIN {X 0.012,Y -195.540,Z 917.841,A 0.000,B 0.000,C 90.000,E1 331.435} C_DIS
LIN {X -0.065,Y -202.072,Z 917.823,A 0.000,B 0.000,C 90.000,E1 328.201} C_DIS
LIN {X -0.006,Y -209.033,Z 917.805,A 0.000,B 0.000,C 90.000,E1 324.975} C_DIS
LIN {X -0.040,Y -216.599,Z 917.788,A 0.000,B 0.000,C 90.000,E1 321.823} C_DIS
LIN {X 0.064,Y -224.687,Z 917.771,A 0.000,B 0.000,C 90.000,E1 318.690} C_DIS
LIN {X 0.035,Y -233.631,Z 917.754,A 0.000,B 0.000,C 90.000,E1 315.648} C_DIS
LIN {X -0.108,Y -243.608,Z 917.737,A 0.000,B 0.000,C 90.000,E1 312.690} C_DIS
LIN {X 0.024,Y -253.299,Z 917.723,A 0.000,B 0.000,C 90.000,E1 310.092} C_DIS
LIN {X -0.063,Y -265.509,Z 917.707,A 0.000,B 0.000,C 90.000,E1 307.237} C_DIS
LIN {X 0.039,Y -275.562,Z 917.695,A 0.000,B 0.000,C 90.000,E1 305.105} C_DIS
LIN {X 0.092,Y -292.209,Z 917.678,A 0.000,B 0.000,C 90.000,E1 302.005} C_DIS
LIN {X 0.020,Y -310.289,Z 917.661,A 0.000,B 0.000,C 90.000,E1 299.027} C_DIS
LIN {X 0.139,Y -325.827,Z 917.649,A 0.000,B 0.000,C 90.000,E1 296.744} C_DIS
LIN {X 0.090,Y -350.609,Z 917.631,A 0.000,B 0.000,C 90.000,E1 293.643} C_DIS
LIN {X -0.098,Y -373.870,Z 917.617,A 0.000,B 0.000,C 90.000,E1 291.099} C_DIS
LIN {X -0.001,Y -386.906,Z 917.609,A 0.000,B 0.000,C 90.000,E1 289.704} C_DIS
LIN {X -0.125,Y -402.472,Z 917.601,A 0.000,B 0.000,C 90.000,E1 288.109} C_DIS
LIN {X 0.213,Y -414.983,Z 917.593,A 0.000,B 0.000,C 90.000,E1 286.732} C_DIS
LIN {X -0.104,Y -427.351,Z 917.586,A 0.000,B 0.000,C 90.000,E1 285.426} C_DIS
LIN {X -0.152,Y -436.727,Z 917.580,A 0.000,B 0.000,C 90.000,E1 284.356} C_DIS
LIN {X -0.196,Y -445.665,Z 917.574,A 0.000,B 0.000,C 90.000,E1 283.300} C_DIS
LIN {X 0.128,Y -456.141,Z 917.566,A 0.000,B 0.000,C 90.000,E1 281.951} C_DIS
LIN {X -0.130,Y -463.909,Z 917.561,A 0.000,B 0.000,C 90.000,E1 280.950} C_DIS
LIN {X -0.087,Y -473.023,Z 917.554,A 0.000,B 0.000,C 90.000,E1 279.670} C_DIS
LIN {X -0.117,Y -477.967,Z 917.549,A 0.000,B 0.000,C 90.000,E1 278.916} C_DIS
LIN {X -0.109,Y -482.255,Z 917.545,A 0.000,B 0.000,C 90.000,E1 278.163} C_DIS
LIN {X -0.059,Y -485.737,Z 917.541,A 0.000,B 0.000,C 90.000,E1 277.409} C_DIS
LIN {X -0.041,Y -488.510,Z 917.537,A 0.000,B 0.000,C 90.000,E1 276.663} C_DIS
LIN {X 0.164,Y -489.936,Z 917.534,A 0.000,B 0.000,C 90.000,E1 276.144} C_DIS
LIN {X -0.108,Y -490.955,Z 917.531,A 0.000,B 0.000,C 90.000,E1 275.682} C_DIS
LIN {X 0.115,Y -491.691,Z 917.529,A 0.000,B 0.000,C 90.000,E1 275.163} C_DIS
LIN {X -0.148,Y -492.004,Z 917.526,A 0.000,B 0.000,C 90.000,E1 274.702} C_DIS
LIN {X 0.045,Y -491.885,Z 917.523,A 0.000,B 0.000,C 90.000,E1 274.188} C_DIS
LIN {X -0.213,Y -491.295,Z 917.521,A 0.000,B 0.000,C 90.000,E1 273.726} C_DIS
LIN {X -0.013,Y -490.295,Z 917.518,A 0.000,B 0.000,C 90.000,E1 273.212} C_DIS
LIN {X 0.210,Y -488.676,Z 917.515,A 0.000,B 0.000,C 90.000,E1 272.694} C_DIS
LIN {X -0.085,Y -486.418,Z 917.512,A 0.000,B 0.000,C 90.000,E1 272.236} C_DIS
LIN {X -0.238,Y -485.065,Z 917.511,A 0.000,B 0.000,C 90.000,E1 272.007} C_DIS
LIN {X -0.051,Y -481.725,Z 917.508,A 0.000,B 0.000,C 90.000,E1 271.489} C_DIS
LIN {X 0.102,Y -477.491,Z 917.505,A 0.000,B 0.000,C 90.000,E1 270.974} C_DIS
LIN {X -0.217,Y -472.333,Z 917.503,A 0.000,B 0.000,C 90.000,E1 270.516} C_DIS
LIN {X 0.182,Y -466.475,Z 917.500,A 0.000,B 0.000,C 90.000,E1 270.000} C_DIS
LIN {X 0.062,Y -460.278,Z 917.498,A 0.000,B 0.000,C 90.000,E1 269.599} C_DIS
LIN {X -0.109,Y -453.642,Z 917.496,A 0.000,B 0.000,C 90.000,E1 269.255} C_DIS
LIN {X 0.126,Y -446.885,Z 917.494,A 0.000,B 0.000,C 90.000,E1 268.912} C_DIS
LIN {X -0.189,Y -440.010,Z 917.493,A 0.000,B 0.000,C 90.000,E1 268.682} C_DIS
LIN {X -0.161,Y -432.824,Z 917.491,A 0.000,B 0.000,C 90.000,E1 268.453} C_DIS
LIN {X 0.181,Y -425.423,Z 917.490,A 0.000,B 0.000,C 90.000,E1 268.224} C_DIS
LIN {X 0.005,Y -416.410,Z 917.490,A 0.000,B 0.000,C 90.000,E1 268.108} C_DIS
LIN {X -0.114,Y -406.500,Z 917.489,A 0.000,B 0.000,C 90.000,E1 268.051} C_DIS
LIN {X -0.171,Y -402.832,Z 917.489,A 0.000,B 0.000,C 90.000,E1 268.051} C_DIS
LIN {X 0.078,Y -181.127,Z 917.489,A 0.000,B 0.000,C 90.000,E1 267.993} C_DIS
LIN {X -0.039,Y -180.906,Z 917.475,A 0.000,B 0.000,C 90.000,E1 265.469} C_DIS
LIN {X 0.019,Y -180.731,Z 917.470,A 0.000,B 0.000,C 90.000,E1 264.609} C_DIS
LIN {X -0.060,Y -178.820,Z 917.442,A 0.000,B 0.000,C 90.000,E1 259.567} C_DIS
LIN {X 0.022,Y -175.865,Z 917.414,A 0.000,B 0.000,C 90.000,E1 254.448} C_DIS
LIN {X 0.071,Y -173.833,Z 917.399,A 0.000,B 0.000,C 90.000,E1 251.873} C_DIS
LIN {X 0.005,Y -171.500,Z 917.380,A 0.000,B 0.000,C 90.000,E1 248.465} C_DIS
LIN {X -0.008,Y -167.728,Z 917.356,A 0.000,B 0.000,C 90.000,E1 244.152} C_DIS
LIN {X 0.009,Y -166.423,Z 917.347,A 0.000,B 0.000,C 90.000,E1 242.410} C_DIS
LIN {X 0.006,Y -163.145,Z 917.327,A 0.000,B 0.000,C 90.000,E1 238.918} C_DIS
LIN {X -0.029,Y -161.099,Z 917.313,A 0.000,B 0.000,C 90.000,E1 236.294} C_DIS
LIN {X -0.045,Y -157.827,Z 917.293,A 0.000,B 0.000,C 90.000,E1 232.763} C_DIS
LIN {X 0.019,Y -155.860,Z 917.278,A 0.000,B 0.000,C 90.000,E1 230.070} C_DIS
LIN {X 0.074,Y -152.110,Z 917.253,A 0.000,B 0.000,C 90.000,E1 225.567} C_DIS
LIN {X -0.018,Y -150.361,Z 917.238,A 0.000,B 0.000,C 90.000,E1 222.894} C_DIS
LIN {X 0.021,Y -147.096,Z 917.213,A 0.000,B 0.000,C 90.000,E1 218.338} C_DIS
LIN {X 0.015,Y -145.666,Z 917.198,A 0.000,B 0.000,C 90.000,E1 215.598} C_DIS
LIN {X 0.019,Y -143.049,Z 917.172,A 0.000,B 0.000,C 90.000,E1 211.003} C_DIS
LIN {X -0.046,Y -141.672,Z 917.152,A 0.000,B 0.000,C 90.000,E1 207.334} C_DIS
LIN {X 0.064,Y -139.452,Z 917.116,A 0.000,B 0.000,C 90.000,E1 200.791} C_DIS
LIN {X -0.016,Y -139.186,Z 917.105,A 0.000,B 0.000,C 90.000,E1 198.960} C_DIS
LIN {X 0.007,Y -138.323,Z 917.053,A 0.000,B 0.000,C 90.000,E1 189.613} C_DIS
LIN {X 0.014,Y -139.460,Z 917.007,A 0.000,B 0.000,C 90.000,E1 181.203} C_DIS
LIN {X -0.046,Y -141.014,Z 916.976,A 0.000,B 0.000,C 90.000,E1 175.641} C_DIS
LIN {X 0.045,Y -142.768,Z 916.955,A 0.000,B 0.000,C 90.000,E1 171.894} C_DIS
LIN {X 0.000,Y -145.178,Z 916.929,A 0.000,B 0.000,C 90.000,E1 167.297} C_DIS
LIN {X 0.034,Y -147.801,Z 916.909,A 0.000,B 0.000,C 90.000,E1 163.614} C_DIS
LIN {X -0.072,Y -150.486,Z 916.889,A 0.000,B 0.000,C 90.000,E1 160.007} C_DIS
LIN {X 0.002,Y -153.941,Z 916.869,A 0.000,B 0.000,C 90.000,E1 156.357} C_DIS
LIN {X 0.065,Y -157.353,Z 916.849,A 0.000,B 0.000,C 90.000,E1 152.743} C_DIS
LIN {X 0.008,Y -161.548,Z 916.829,A 0.000,B 0.000,C 90.000,E1 149.203} C_DIS
LIN {X 0.020,Y -165.746,Z 916.809,A 0.000,B 0.000,C 90.000,E1 145.674} C_DIS
LIN {X 0.007,Y -170.700,Z 916.790,A 0.000,B 0.000,C 90.000,E1 142.190} C_DIS
LIN {X -0.081,Y -175.573,Z 916.771,A 0.000,B 0.000,C 90.000,E1 138.771} C_DIS
LIN {X 0.038,Y -181.191,Z 916.752,A 0.000,B 0.000,C 90.000,E1 135.324} C_DIS
LIN {X -0.094,Y -186.652,Z 916.733,A 0.000,B 0.000,C 90.000,E1 132.000} C_DIS
LIN {X -0.024,Y -191.257,Z 916.719,A 0.000,B 0.000,C 90.000,E1 129.483} C_DIS
LIN {X 0.039,Y -193.775,Z 916.711,A 0.000,B 0.000,C 90.000,E1 127.971} C_DIS
LIN {X 0.025,Y -295.545,Z 916.711,A 0.000,B 0.000,C 90.000,E1 127.971} C_DIS
LIN {X -0.081,Y -297.062,Z 916.711,A 0.000,B 0.000,C 90.000,E1 127.971} C_DIS
LIN {X 0.087,Y -300.501,Z 916.710,A 0.000,B 0.000,C 90.000,E1 127.810} C_DIS
LIN {X -0.065,Y -303.747,Z 916.709,A 0.000,B 0.000,C 90.000,E1 127.604} C_DIS
LIN {X 0.011,Y -307.429,Z 916.706,A 0.000,B 0.000,C 90.000,E1 127.156} C_DIS
LIN {X -0.162,Y -309.323,Z 916.705,A 0.000,B 0.000,C 90.000,E1 126.870} C_DIS
LIN {X 0.098,Y -310.805,Z 916.703,A 0.000,B 0.000,C 90.000,E1 126.503} C_DIS
LIN {X -0.073,Y -312.977,Z 916.699,A 0.000,B 0.000,C 90.000,E1 125.884} C_DIS
LIN {X -0.111,Y -323.342,Z 916.681,A 0.000,B 0.000,C 90.000,E1 122.673} C_DIS
LIN {X 0.094,Y -334.009,Z 916.666,A 0.000,B 0.000,C 90.000,E1 119.795} C_DIS
LIN {X 0.118,Y -346.048,Z 916.650,A 0.000,B 0.000,C 90.000,E1 117.001} C_DIS
LIN {X 0.033,Y -359.560,Z 916.635,A 0.000,B 0.000,C 90.000,E1 114.283} C_DIS
LIN {X 0.087,Y -372.907,Z 916.622,A 0.000,B 0.000,C 90.000,E1 111.897} C_DIS
LIN {X 0.054,Y -387.609,Z 916.609,A 0.000,B 0.000,C 90.000,E1 109.577} C_DIS
LIN {X -0.119,Y -403.773,Z 916.596,A 0.000,B 0.000,C 90.000,E1 107.330} C_DIS
LIN {X 0.142,Y -421.513,Z 916.584,A 0.000,B 0.000,C 90.000,E1 105.079} C_DIS
LIN {X 0.095,Y -440.878,Z 916.572,A 0.000,B 0.000,C 90.000,E1 102.939} C_DIS
LIN {X 0.043,Y -461.095,Z 916.561,A 0.000,B 0.000,C 90.000,E1 100.950} C_DIS
LIN {X -0.051,Y -466.235,Z 916.558,A 0.000,B 0.000,C 90.000,E1 100.489} C_DIS
LIN {X -0.034,Y -468.539,Z 916.557,A 0.000,B 0.000,C 90.000,E1 100.254} C_DIS
LIN {X -0.153,Y -470.378,Z 916.556,A 0.000,B 0.000,C 90.000,E1 100.018} C_DIS
LIN {X 0.192,Y -471.765,Z 916.554,A 0.000,B 0.000,C 90.000,E1 99.726} C_DIS
LIN {X -0.176,Y -473.556,Z 916.551,A 0.000,B 0.000,C 90.000,E1 99.265} C_DIS
LIN {X -0.068,Y -474.261,Z 916.549,A 0.000,B 0.000,C 90.000,E1 98.746} C_DIS
LIN {X 0.124,Y -473.997,Z 916.546,A 0.000,B 0.000,C 90.000,E1 98.219} C_DIS
LIN {X -0.220,Y -472.733,Z 916.543,A 0.000,B 0.000,C 90.000,E1 97.757} C_DIS
LIN {X 0.046,Y -471.664,Z 916.542,A 0.000,B 0.000,C 90.000,E1 97.473} C_DIS
LIN {X 0.223,Y -468.555,Z 916.539,A 0.000,B 0.000,C 90.000,E1 96.947} C_DIS
LIN {X 0.039,Y -449.546,Z 916.522,A 0.000,B 0.000,C 90.000,E1 93.898} C_DIS
LIN {X -0.107,Y -440.103,Z 916.513,A 0.000,B 0.000,C 90.000,E1 92.350} C_DIS
LIN {X 0.024,Y -430.436,Z 916.504,A 0.000,B 0.000,C 90.000,E1 90.745} C_DIS
LIN {X -0.110,Y -416.042,Z 916.491,A 0.000,B 0.000,C 90.000,E1 88.339} C_DIS
LIN {X 0.097,Y -404.996,Z 916.480,A 0.000,B 0.000,C 90.000,E1 86.388} C_DIS
LIN {X 0.109,Y -393.950,Z 916.469,A 0.000,B 0.000,C 90.000,E1 84.432} C_DIS
LIN {X -0.065,Y -382.910,Z 916.458,A 0.000,B 0.000,C 90.000,E1 82.470} C_DIS
LIN {X -0.043,Y -373.358,Z 916.448,A 0.000,B 0.000,C 90.000,E1 80.735} C_DIS
LIN {X -0.140,Y -363.609,Z 916.439,A 0.000,B 0.000,C 90.000,E1 78.993} C_DIS
LIN {X 0.030,Y -351.939,Z 916.427,A 0.000,B 0.000,C 90.000,E1 76.881} C_DIS
LIN {X -0.077,Y -337.053,Z 916.412,A 0.000,B 0.000,C 90.000,E1 74.157} C_DIS
LIN {X 0.130,Y -320.176,Z 916.393,A 0.000,B 0.000,C 90.000,E1 70.678} C_DIS
LIN {X -0.042,Y -309.759,Z 916.380,A 0.000,B 0.000,C 90.000,E1 68.465} C_DIS
LIN {X -0.025,Y -299.441,Z 916.368,A 0.000,B 0.000,C 90.000,E1 66.177} C_DIS
LIN {X -0.003,Y -289.085,Z 916.355,A 0.000,B 0.000,C 90.000,E1 63.845} C_DIS
LIN {X -0.030,Y -280.067,Z 916.343,A 0.000,B 0.000,C 90.000,E1 61.820} C_DIS
LIN {X -0.110,Y -268.164,Z 916.328,A 0.000,B 0.000,C 90.000,E1 59.076} C_DIS
LIN {X -0.045,Y -255.196,Z 916.310,A 0.000,B 0.000,C 90.000,E1 55.881} C_DIS
LIN {X 0.018,Y -246.039,Z 916.296,A 0.000,B 0.000,C 90.000,E1 53.336} C_DIS
LIN {X -0.045,Y -235.556,Z 916.278,A 0.000,B 0.000,C 90.000,E1 50.033} C_DIS
LIN {X -0.034,Y -226.901,Z 916.261,A 0.000,B 0.000,C 90.000,E1 47.025} C_DIS
LIN {X 0.054,Y -218.899,Z 916.244,A 0.000,B 0.000,C 90.000,E1 43.947} C_DIS
LIN {X -0.033,Y -211.247,Z 916.227,A 0.000,B 0.000,C 90.000,E1 40.862} C_DIS
LIN {X 0.042,Y -204.465,Z 916.209,A 0.000,B 0.000,C 90.000,E1 37.684} C_DIS
LIN {X 0.023,Y -198.090,Z 916.192,A 0.000,B 0.000,C 90.000,E1 34.485} C_DIS
LIN {X -0.055,Y -192.123,Z 916.174,A 0.000,B 0.000,C 90.000,E1 31.258} C_DIS
LIN {X -0.080,Y -186.799,Z 916.155,A 0.000,B 0.000,C 90.000,E1 27.975} C_DIS
LIN {X -0.077,Y -182.089,Z 916.137,A 0.000,B 0.000,C 90.000,E1 24.643} C_DIS
LIN {X 0.079,Y -178.062,Z 916.118,A 0.000,B 0.000,C 90.000,E1 21.227} C_DIS
LIN {X 0.050,Y -173.995,Z 916.094,A 0.000,B 0.000,C 90.000,E1 16.985} C_DIS
LIN {X 0.073,Y -170.630,Z 916.066,A 0.000,B 0.000,C 90.000,E1 11.827} C_DIS
LIN {X -0.015,Y -168.419,Z 916.027,A 0.000,B 0.000,C 90.000,E1 4.935} C_DIS
LIN {X 0.048,Y -169.751,Z 915.973,A 0.000,B 0.000,C 90.000,E1 355.179} C_DIS
LIN {X -0.079,Y -172.516,Z 915.945,A 0.000,B 0.000,C 90.000,E1 350.038} C_DIS
LIN {X 0.065,Y -175.930,Z 915.921,A 0.000,B 0.000,C 90.000,E1 345.700} C_DIS
LIN {X 0.029,Y -180.319,Z 915.897,A 0.000,B 0.000,C 90.000,E1 341.456} C_DIS
LIN {X -0.031,Y -184.628,Z 915.878,A 0.000,B 0.000,C 90.000,E1 338.103} C_DIS
LIN {X -0.045,Y -189.848,Z 915.860,A 0.000,B 0.000,C 90.000,E1 334.768} C_DIS
LIN {X 0.073,Y -195.852,Z 915.841,A 0.000,B 0.000,C 90.000,E1 331.435} C_DIS
LIN {X 0.005,Y -202.359,Z 915.823,A 0.000,B 0.000,C 90.000,E1 328.201} C_DIS
LIN {X 0.074,Y -209.328,Z 915.806,A 0.000,B 0.000,C 90.000,E1 324.975} C_DIS
LIN {X 0.050,Y -216.863,Z 915.788,A 0.000,B 0.000,C 90.000,E1 321.823} C_DIS
LIN {X 0.017,Y -224.938,Z 915.771,A 0.000,B 0.000,C 90.000,E1 318.728} C_DIS
LIN {X -0.017,Y -233.898,Z 915.754,A 0.000,B 0.000,C 90.000,E1 315.688} C_DIS
LIN {X 0.016,Y -243.852,Z 915.737,A 0.000,B 0.000,C 90.000,E1 312.690} C_DIS
LIN {X -0.022,Y -254.988,Z 915.721,A 0.000,B 0.000,C 90.000,E1 309.769} C_DIS
LIN {X 0.139,Y -267.266,Z 915.705,A 0.000,B 0.000,C 90.000,E1 306.870} C_DIS
LIN {X -0.071,Y -281.021,Z 915.689,A 0.000,B 0.000,C 90.000,E1 304.119} C_DIS
LIN {X -0.021,Y -298.055,Z 915.672,A 0.000,B 0.000,C 90.000,E1 301.052} C_DIS
LIN {X -0.039,Y -312.355,Z 915.660,A 0.000,B 0.000,C 90.000,E1 298.743} C_DIS
LIN {X 0.033,Y -325.648,Z 915.649,A 0.000,B 0.000,C 90.000,E1 296.796} C_DIS
LIN {X -0.092,Y -347.777,Z 915.633,A 0.000,B 0.000,C 90.000,E1 294.003} C_DIS
LIN {X -0.056,Y -371.271,Z 915.619,A 0.000,B 0.000,C 90.000,E1 291.354} C_DIS
LIN {X 0.102,Y -386.615,Z 915.610,A 0.000,B 0.000,C 90.000,E1 289.704} C_DIS
LIN {X -0.068,Y -402.201,Z 915.601,A 0.000,B 0.000,C 90.000,E1 288.109} C_DIS
LIN {X -0.251,Y -414.722,Z 915.593,A 0.000,B 0.000,C 90.000,E1 286.804} C_DIS
LIN {X -0.028,Y -427.077,Z 915.586,A 0.000,B 0.000,C 90.000,E1 285.426} C_DIS
LIN {X -0.077,Y -436.489,Z 915.580,A 0.000,B 0.000,C 90.000,E1 284.356} C_DIS
LIN {X -0.123,Y -445.467,Z 915.574,A 0.000,B 0.000,C 90.000,E1 283.300} C_DIS
LIN {X -0.058,Y -453.939,Z 915.568,A 0.000,B 0.000,C 90.000,E1 282.243} C_DIS
LIN {X 0.109,Y -461.856,Z 915.562,A 0.000,B 0.000,C 90.000,E1 281.186} C_DIS
LIN {X 0.136,Y -471.103,Z 915.555,A 0.000,B 0.000,C 90.000,E1 279.905} C_DIS
LIN {X 0.088,Y -476.290,Z 915.551,A 0.000,B 0.000,C 90.000,E1 279.151} C_DIS
LIN {X 0.092,Y -480.834,Z 915.547,A 0.000,B 0.000,C 90.000,E1 278.398} C_DIS
LIN {X 0.129,Y -484.607,Z 915.543,A 0.000,B 0.000,C 90.000,E1 277.644} C_DIS
LIN {X -0.169,Y -486.720,Z 915.540,A 0.000,B 0.000,C 90.000,E1 277.182} C_DIS
LIN {X 0.029,Y -488.513,Z 915.537,A 0.000,B 0.000,C 90.000,E1 276.663} C_DIS
LIN {X -0.252,Y -489.905,Z 915.534,A 0.000,B 0.000,C 90.000,E1 276.201} C_DIS
LIN {X -0.037,Y -490.980,Z 915.532,A 0.000,B 0.000,C 90.000,E1 275.682} C_DIS
LIN {X 0.186,Y -491.682,Z 915.529,A 0.000,B 0.000,C 90.000,E1 275.163} C_DIS
LIN {X -0.076,Y -492.049,Z 915.526,A 0.000,B 0.000,C 90.000,E1 274.702} C_DIS
LIN {X 0.116,Y -491.959,Z 915.523,A 0.000,B 0.000,C 90.000,E1 274.188} C_DIS
LIN {X -0.142,Y -491.409,Z 915.521,A 0.000,B 0.000,C 90.000,E1 273.726} C_DIS
LIN {X 0.058,Y -490.395,Z 915.518,A 0.000,B 0.000,C 90.000,E1 273.212} C_DIS
LIN {X -0.207,Y -488.793,Z 915.515,A 0.000,B 0.000,C 90.000,E1 272.751} C_DIS
LIN {X -0.013,Y -486.604,Z 915.512,A 0.000,B 0.000,C 90.000,E1 272.236} C_DIS
LIN {X 0.182,Y -483.695,Z 915.510,A 0.000,B 0.000,C 90.000,E1 271.718} C_DIS
LIN {X -0.136,Y -480.038,Z 915.507,A 0.000,B 0.000,C 90.000,E1 271.260} C_DIS
LIN {X 0.009,Y -475.405,Z 915.504,A 0.000,B 0.000,C 90.000,E1 270.745} C_DIS
LIN {X -0.155,Y -472.731,Z 915.503,A 0.000,B 0.000,C 90.000,E1 270.516} C_DIS
LIN {X 0.228,Y -466.910,Z 915.500,A 0.000,B 0.000,C 90.000,E1 270.000} C_DIS
LIN {X -0.162,Y -463.877,Z 915.499,A 0.000,B 0.000,C 90.000,E1 269.828} C_DIS
LIN {X -0.149,Y -457.357,Z 915.497,A 0.000,B 0.000,C 90.000,E1 269.427} C_DIS
LIN {X -0.131,Y -450.615,Z 915.495,A 0.000,B 0.000,C 90.000,E1 269.083} C_DIS
LIN {X -0.163,Y -443.929,Z 915.493,A 0.000,B 0.000,C 90.000,E1 268.797} C_DIS
LIN {X 0.086,Y -436.712,Z 915.492,A 0.000,B 0.000,C 90.000,E1 268.511} C_DIS
LIN {X -0.168,Y -429.486,Z 915.491,A 0.000,B 0.000,C 90.000,E1 268.339} C_DIS
LIN {X -0.125,Y -421.171,Z 915.490,A 0.000,B 0.000,C 90.000,E1 268.165} C_DIS
LIN {X 0.057,Y -413.523,Z 915.489,A 0.000,B 0.000,C 90.000,E1 268.051} C_DIS
LIN {X 0.133,Y -406.094,Z 915.489,A 0.000,B 0.000,C 90.000,E1 267.993} C_DIS
LIN {X 0.033,Y -181.125,Z 915.489,A 0.000,B 0.000,C 90.000,E1 267.993} C_DIS
LIN {X 0.071,Y -180.907,Z 915.475,A 0.000,B 0.000,C 90.000,E1 265.412} C_DIS
LIN {X -0.053,Y -180.720,Z 915.470,A 0.000,B 0.000,C 90.000,E1 264.609} C_DIS
LIN {X 0.046,Y -178.809,Z 915.442,A 0.000,B 0.000,C 90.000,E1 259.511} C_DIS
LIN {X -0.048,Y -175.854,Z 915.414,A 0.000,B 0.000,C 90.000,E1 254.448} C_DIS
LIN {X -0.065,Y -173.180,Z 915.395,A 0.000,B 0.000,C 90.000,E1 251.040} C_DIS
LIN {X -0.063,Y -171.481,Z 915.380,A 0.000,B 0.000,C 90.000,E1 248.465} C_DIS
LIN {X -0.075,Y -167.711,Z 915.356,A 0.000,B 0.000,C 90.000,E1 244.152} C_DIS
LIN {X -0.059,Y -166.401,Z 915.347,A 0.000,B 0.000,C 90.000,E1 242.410} C_DIS
LIN {X 0.079,Y -163.126,Z 915.327,A 0.000,B 0.000,C 90.000,E1 238.869} C_DIS
LIN {X -0.094,Y -161.077,Z 915.313,A 0.000,B 0.000,C 90.000,E1 236.294} C_DIS
LIN {X 0.017,Y -157.808,Z 915.293,A 0.000,B 0.000,C 90.000,E1 232.718} C_DIS
LIN {X -0.045,Y -155.844,Z 915.278,A 0.000,B 0.000,C 90.000,E1 230.070} C_DIS
LIN {X 0.010,Y -152.093,Z 915.253,A 0.000,B 0.000,C 90.000,E1 225.567} C_DIS
LIN {X 0.029,Y -150.344,Z 915.238,A 0.000,B 0.000,C 90.000,E1 222.852} C_DIS
LIN {X 0.051,Y -147.082,Z 915.213,A 0.000,B 0.000,C 90.000,E1 218.302} C_DIS
LIN {X -0.047,Y -145.655,Z 915.198,A 0.000,B 0.000,C 90.000,E1 215.598} C_DIS
LIN {X -0.042,Y -143.038,Z 915.172,A 0.000,B 0.000,C 90.000,E1 211.003} C_DIS
LIN {X -0.042,Y -141.661,Z 915.152,A 0.000,B 0.000,C 90.000,E1 207.308} C_DIS
LIN {X 0.003,Y -139.449,Z 915.116,A 0.000,B 0.000,C 90.000,E1 200.791} C_DIS
LIN {X 0.056,Y -139.182,Z 915.105,A 0.000,B 0.000,C 90.000,E1 198.906} C_DIS
LIN {X -0.052,Y -138.321,Z 915.053,A 0.000,B 0.000,C 90.000,E1 189.613} C_DIS
LIN {X -0.046,Y -139.464,Z 915.007,A 0.000,B 0.000,C 90.000,E1 181.203} C_DIS
LIN {X 0.034,Y -141.025,Z 914.976,A 0.000,B 0.000,C 90.000,E1 175.584} C_DIS
LIN {X -0.011,Y -142.391,Z 914.960,A 0.000,B 0.000,C 90.000,E1 172.818} C_DIS
LIN {X 0.052,Y -144.621,Z 914.934,A 0.000,B 0.000,C 90.000,E1 168.173} C_DIS
LIN {X -0.029,Y -147.816,Z 914.909,A 0.000,B 0.000,C 90.000,E1 163.614} C_DIS
LIN {X 0.058,Y -150.505,Z 914.889,A 0.000,B 0.000,C 90.000,E1 159.934} C_DIS
LIN {X -0.063,Y -153.965,Z 914.869,A 0.000,B 0.000,C 90.000,E1 156.357} C_DIS
LIN {X 0.000,Y -157.377,Z 914.849,A 0.000,B 0.000,C 90.000,E1 152.743} C_DIS
LIN {X -0.058,Y -161.579,Z 914.829,A 0.000,B 0.000,C 90.000,E1 149.203} C_DIS
LIN {X -0.047,Y -165.776,Z 914.809,A 0.000,B 0.000,C 90.000,E1 145.674} C_DIS
LIN {X -0.061,Y -170.735,Z 914.790,A 0.000,B 0.000,C 90.000,E1 142.190} C_DIS
LIN {X -0.019,Y -175.608,Z 914.771,A 0.000,B 0.000,C 90.000,E1 138.728} C_DIS
LIN {X -0.033,Y -181.224,Z 914.752,A 0.000,B 0.000,C 90.000,E1 135.324} C_DIS
LIN {X 0.099,Y -186.691,Z 914.733,A 0.000,B 0.000,C 90.000,E1 131.919} C_DIS
LIN {X 0.051,Y -191.292,Z 914.719,A 0.000,B 0.000,C 90.000,E1 129.439} C_DIS
LIN {X -0.043,Y -193.738,Z 914.711,A 0.000,B 0.000,C 90.000,E1 128.016} C_DIS
LIN {X -0.101,Y -295.673,Z 914.711,A 0.000,B 0.000,C 90.000,E1 128.016} C_DIS
LIN {X -0.028,Y -301.171,Z 914.710,A 0.000,B 0.000,C 90.000,E1 127.810} C_DIS
LIN {X -0.010,Y -304.158,Z 914.709,A 0.000,B 0.000,C 90.000,E1 127.569} C_DIS
LIN {X 0.114,Y -307.889,Z 914.706,A 0.000,B 0.000,C 90.000,E1 127.076} C_DIS
LIN {X -0.112,Y -309.709,Z 914.704,A 0.000,B 0.000,C 90.000,E1 126.790} C_DIS
LIN {X -0.090,Y -311.129,Z 914.702,A 0.000,B 0.000,C 90.000,E1 126.457} C_DIS
LIN {X -0.076,Y -313.194,Z 914.699,A 0.000,B 0.000,C 90.000,E1 125.804} C_DIS
LIN {X 0.162,Y -323.598,Z 914.681,A 0.000,B 0.000,C 90.000,E1 122.546} C_DIS
LIN {X -0.070,Y -334.301,Z 914.665,A 0.000,B 0.000,C 90.000,E1 119.745} C_DIS
LIN {X -0.035,Y -346.379,Z 914.650,A 0.000,B 0.000,C 90.000,E1 116.950} C_DIS
LIN {X 0.040,Y -359.932,Z 914.635,A 0.000,B 0.000,C 90.000,E1 114.207} C_DIS
LIN {X -0.044,Y -373.320,Z 914.621,A 0.000,B 0.000,C 90.000,E1 111.844} C_DIS
LIN {X 0.064,Y -388.066,Z 914.608,A 0.000,B 0.000,C 90.000,E1 109.504} C_DIS
LIN {X 0.159,Y -404.277,Z 914.596,A 0.000,B 0.000,C 90.000,E1 107.221} C_DIS
LIN {X 0.156,Y -422.068,Z 914.583,A 0.000,B 0.000,C 90.000,E1 105.009} C_DIS
LIN {X 0.023,Y -441.474,Z 914.572,A 0.000,B 0.000,C 90.000,E1 102.883} C_DIS
LIN {X 0.014,Y -461.709,Z 914.561,A 0.000,B 0.000,C 90.000,E1 100.894} C_DIS
LIN {X -0.069,Y -466.848,Z 914.558,A 0.000,B 0.000,C 90.000,E1 100.433} C_DIS
LIN {X -0.047,Y -468.995,Z 914.557,A 0.000,B 0.000,C 90.000,E1 100.197} C_DIS
LIN {X -0.200,Y -470.748,Z 914.555,A 0.000,B 0.000,C 90.000,E1 99.962} C_DIS
LIN {X 0.110,Y -472.064,Z 914.554,A 0.000,B 0.000,C 90.000,E1 99.670} C_DIS
LIN {X 0.213,Y -473.706,Z 914.551,A 0.000,B 0.000,C 90.000,E1 99.151} C_DIS
LIN {X -0.072,Y -474.287,Z 914.548,A 0.000,B 0.000,C 90.000,E1 98.681} C_DIS
LIN {X 0.049,Y -473.905,Z 914.545,A 0.000,B 0.000,C 90.000,E1 98.163} C_DIS
LIN {X 0.174,Y -472.504,Z 914.543,A 0.000,B 0.000,C 90.000,E1 97.644} C_DIS
LIN {X 0.033,Y -471.352,Z 914.541,A 0.000,B 0.000,C 90.000,E1 97.409} C_DIS
LIN {X 0.107,Y -460.066,Z 914.531,A 0.000,B 0.000,C 90.000,E1 95.625} C_DIS
LIN {X 0.163,Y -447.652,Z 914.520,A 0.000,B 0.000,C 90.000,E1 93.555} C_DIS
LIN {X 0.169,Y -436.555,Z 914.510,A 0.000,B 0.000,C 90.000,E1 91.718} C_DIS
LIN {X 0.059,Y -423.648,Z 914.498,A 0.000,B 0.000,C 90.000,E1 89.599} C_DIS
LIN {X 0.085,Y -410.963,Z 914.486,A 0.000,B 0.000,C 90.000,E1 87.421} C_DIS
LIN {X 0.189,Y -399.884,Z 914.475,A 0.000,B 0.000,C 90.000,E1 85.469} C_DIS
LIN {X 0.085,Y -388.833,Z 914.464,A 0.000,B 0.000,C 90.000,E1 83.514} C_DIS
LIN {X -0.145,Y -377.772,Z 914.453,A 0.000,B 0.000,C 90.000,E1 81.546} C_DIS
LIN {X -0.156,Y -368.130,Z 914.443,A 0.000,B 0.000,C 90.000,E1 79.803} C_DIS
LIN {X 0.080,Y -358.230,Z 914.433,A 0.000,B 0.000,C 90.000,E1 77.993} C_DIS
LIN {X 0.126,Y -346.553,Z 914.422,A 0.000,B 0.000,C 90.000,E1 75.880} C_DIS
LIN {X 0.132,Y -328.884,Z 914.403,A 0.000,B 0.000,C 90.000,E1 72.489} C_DIS
LIN {X -0.135,Y -316.868,Z 914.389,A 0.000,B 0.000,C 90.000,E1 70.007} C_DIS
LIN {X -0.055,Y -305.039,Z 914.374,A 0.000,B 0.000,C 90.000,E1 67.411} C_DIS
LIN {X -0.026,Y -294.704,Z 914.362,A 0.000,B 0.000,C 90.000,E1 65.101} C_DIS
LIN {X -0.056,Y -287.307,Z 914.352,A 0.000,B 0.000,C 90.000,E1 63.435} C_DIS
LIN {X 0.006,Y -278.290,Z 914.341,A 0.000,B 0.000,C 90.000,E1 61.385} C_DIS
LIN {X 0.010,Y -266.437,Z 914.326,A 0.000,B 0.000,C 90.000,E1 58.614} C_DIS
LIN {X 0.155,Y -253.606,Z 914.308,A 0.000,B 0.000,C 90.000,E1 55.388} C_DIS
LIN {X -0.014,Y -244.660,Z 914.294,A 0.000,B 0.000,C 90.000,E1 52.889} C_DIS
LIN {X 0.067,Y -234.322,Z 914.275,A 0.000,B 0.000,C 90.000,E1 49.542} C_DIS
LIN {X 0.125,Y -224.783,Z 914.256,A 0.000,B 0.000,C 90.000,E1 46.134} C_DIS
LIN {X 0.008,Y -216.919,Z 914.239,A 0.000,B 0.000,C 90.000,E1 43.095} C_DIS
LIN {X 0.035,Y -209.446,Z 914.222,A 0.000,B 0.000,C 90.000,E1 39.967} C_DIS
LIN {X 0.061,Y -202.886,Z 914.204,A 0.000,B 0.000,C 90.000,E1 36.790} C_DIS
LIN {X 0.044,Y -196.560,Z 914.187,A 0.000,B 0.000,C 90.000,E1 33.579} C_DIS
LIN {X -0.011,Y -190.799,Z 914.169,A 0.000,B 0.000,C 90.000,E1 30.335} C_DIS
LIN {X 0.095,Y -185.659,Z 914.150,A 0.000,B 0.000,C 90.000,E1 27.001} C_DIS
LIN {X -0.015,Y -181.139,Z 914.132,A 0.000,B 0.000,C 90.000,E1 23.695} C_DIS
LIN {X 0.046,Y -177.292,Z 914.113,A 0.000,B 0.000,C 90.000,E1 20.301} C_DIS
LIN {X -0.063,Y -173.495,Z 914.089,A 0.000,B 0.000,C 90.000,E1 16.079} C_DIS
LIN {X 0.025,Y -170.417,Z 914.061,A 0.000,B 0.000,C 90.000,E1 10.894} C_DIS
LIN {X 0.055,Y -168.557,Z 914.017,A 0.000,B 0.000,C 90.000,E1 3.094} C_DIS
LIN {X 0.045,Y -170.381,Z 913.969,A 0.000,B 0.000,C 90.000,E1 354.318} C_DIS
LIN {X -0.012,Y -173.405,Z 913.940,A 0.000,B 0.000,C 90.000,E1 349.162} C_DIS
LIN {X 0.033,Y -176.987,Z 913.916,A 0.000,B 0.000,C 90.000,E1 344.866} C_DIS
LIN {X 0.066,Y -180.583,Z 913.897,A 0.000,B 0.000,C 90.000,E1 341.456} C_DIS
LIN {X 0.013,Y -184.919,Z 913.878,A 0.000,B 0.000,C 90.000,E1 338.103} C_DIS
LIN {X -0.074,Y -190.156,Z 913.860,A 0.000,B 0.000,C 90.000,E1 334.793} C_DIS
LIN {X 0.041,Y -196.147,Z 913.842,A 0.000,B 0.000,C 90.000,E1 331.463} C_DIS
LIN {X 0.077,Y -202.643,Z 913.823,A 0.000,B 0.000,C 90.000,E1 328.201} C_DIS
LIN {X -0.017,Y -209.614,Z 913.806,A 0.000,B 0.000,C 90.000,E1 325.022} C_DIS
LIN {X 0.007,Y -217.132,Z 913.788,A 0.000,B 0.000,C 90.000,E1 321.859} C_DIS
LIN {X -0.117,Y -226.275,Z 913.769,A 0.000,B 0.000,C 90.000,E1 318.405} C_DIS
LIN {X 0.047,Y -235.338,Z 913.752,A 0.000,B 0.000,C 90.000,E1 315.324} C_DIS
LIN {X -0.053,Y -245.409,Z 913.735,A 0.000,B 0.000,C 90.000,E1 312.366} C_DIS
LIN {X -0.022,Y -256.667,Z 913.719,A 0.000,B 0.000,C 90.000,E1 309.439} C_DIS
LIN {X -0.020,Y -269.052,Z 913.703,A 0.000,B 0.000,C 90.000,E1 306.583} C_DIS
LIN {X 0.041,Y -282.955,Z 913.688,A 0.000,B 0.000,C 90.000,E1 303.785} C_DIS
LIN {X -0.002,Y -300.040,Z 913.671,A 0.000,B 0.000,C 90.000,E1 300.747} C_DIS
LIN {X 0.042,Y -314.394,Z 913.658,A 0.000,B 0.000,C 90.000,E1 298.437} C_DIS
LIN {X 0.163,Y -327.819,Z 913.647,A 0.000,B 0.000,C 90.000,E1 296.488} C_DIS
LIN {X -0.027,Y -347.467,Z 913.633,A 0.000,B 0.000,C 90.000,E1 294.027} C_DIS
LIN {X -0.108,Y -371.194,Z 913.619,A 0.000,B 0.000,C 90.000,E1 291.354} C_DIS
LIN {X 0.025,Y -386.552,Z 913.609,A 0.000,B 0.000,C 90.000,E1 289.704} C_DIS
LIN {X 0.107,Y -402.291,Z 913.600,A 0.000,B 0.000,C 90.000,E1 288.055} C_DIS
LIN {X -0.003,Y -414.870,Z 913.593,A 0.000,B 0.000,C 90.000,E1 286.732} C_DIS
LIN {X -0.090,Y -424.838,Z 913.587,A 0.000,B 0.000,C 90.000,E1 285.662} C_DIS
LIN {X 0.084,Y -432.066,Z 913.582,A 0.000,B 0.000,C 90.000,E1 284.828} C_DIS
LIN {X -0.230,Y -443.492,Z 913.575,A 0.000,B 0.000,C 90.000,E1 283.536} C_DIS
LIN {X -0.191,Y -452.087,Z 913.569,A 0.000,B 0.000,C 90.000,E1 282.479} C_DIS
LIN {X -0.047,Y -460.152,Z 913.563,A 0.000,B 0.000,C 90.000,E1 281.422} C_DIS
LIN {X -0.052,Y -469.554,Z 913.556,A 0.000,B 0.000,C 90.000,E1 280.141} C_DIS
LIN {X -0.252,Y -476.522,Z 913.551,A 0.000,B 0.000,C 90.000,E1 279.151} C_DIS
LIN {X -0.051,Y -479.621,Z 913.548,A 0.000,B 0.000,C 90.000,E1 278.624} C_DIS
LIN {X -0.024,Y -483.630,Z 913.544,A 0.000,B 0.000,C 90.000,E1 277.871} C_DIS
LIN {X -0.029,Y -486.892,Z 913.540,A 0.000,B 0.000,C 90.000,E1 277.125} C_DIS
LIN {X 0.172,Y -488.628,Z 913.537,A 0.000,B 0.000,C 90.000,E1 276.606} C_DIS
LIN {X -0.108,Y -490.038,Z 913.534,A 0.000,B 0.000,C 90.000,E1 276.144} C_DIS
LIN {X 0.108,Y -491.075,Z 913.531,A 0.000,B 0.000,C 90.000,E1 275.625} C_DIS
LIN {X -0.157,Y -491.753,Z 913.529,A 0.000,B 0.000,C 90.000,E1 275.163} C_DIS
LIN {X 0.071,Y -492.083,Z 913.526,A 0.000,B 0.000,C 90.000,E1 274.645} C_DIS
LIN {X -0.226,Y -491.973,Z 913.523,A 0.000,B 0.000,C 90.000,E1 274.188} C_DIS
LIN {X 0.007,Y -491.399,Z 913.520,A 0.000,B 0.000,C 90.000,E1 273.669} C_DIS
LIN {X 0.208,Y -490.337,Z 913.518,A 0.000,B 0.000,C 90.000,E1 273.154} C_DIS
LIN {X -0.058,Y -488.739,Z 913.515,A 0.000,B 0.000,C 90.000,E1 272.694} C_DIS
LIN {X 0.136,Y -486.538,Z 913.512,A 0.000,B 0.000,C 90.000,E1 272.178} C_DIS
LIN {X -0.154,Y -483.630,Z 913.509,A 0.000,B 0.000,C 90.000,E1 271.718} C_DIS
LIN {X 0.009,Y -479.924,Z 913.507,A 0.000,B 0.000,C 90.000,E1 271.203} C_DIS
LIN {X 0.152,Y -475.263,Z 913.504,A 0.000,B 0.000,C 90.000,E1 270.688} C_DIS
LIN {X -0.153,Y -469.649,Z 913.501,A 0.000,B 0.000,C 90.000,E1 270.229} C_DIS
LIN {X -0.021,Y -463.673,Z 913.499,A 0.000,B 0.000,C 90.000,E1 269.771} C_DIS
LIN {X 0.013,Y -457.163,Z 913.497,A 0.000,B 0.000,C 90.000,E1 269.370} C_DIS
LIN {X 0.029,Y -450.416,Z 913.495,A 0.000,B 0.000,C 90.000,E1 269.026} C_DIS
LIN {X 0.017,Y -443.804,Z 913.493,A 0.000,B 0.000,C 90.000,E1 268.740} C_DIS
LIN {X -0.171,Y -436.595,Z 913.492,A 0.000,B 0.000,C 90.000,E1 268.511} C_DIS
LIN {X 0.015,Y -429.207,Z 913.490,A 0.000,B 0.000,C 90.000,E1 268.282} C_DIS
LIN {X 0.082,Y -420.861,Z 913.490,A 0.000,B 0.000,C 90.000,E1 268.108} C_DIS
LIN {X -0.127,Y -413.251,Z 913.489,A 0.000,B 0.000,C 90.000,E1 268.051} C_DIS
LIN {X -0.035,Y -405.390,Z 913.489,A 0.000,B 0.000,C 90.000,E1 267.993} C_DIS
LIN {X -0.041,Y -181.122,Z 913.489,A 0.000,B 0.000,C 90.000,E1 267.993} C_DIS
LIN {X 0.000,Y -180.907,Z 913.474,A 0.000,B 0.000,C 90.000,E1 265.412} C_DIS
LIN {X 0.057,Y -180.710,Z 913.470,A 0.000,B 0.000,C 90.000,E1 264.552} C_DIS
LIN {X -0.025,Y -178.796,Z 913.442,A 0.000,B 0.000,C 90.000,E1 259.511} C_DIS
LIN {X 0.052,Y -175.842,Z 913.413,A 0.000,B 0.000,C 90.000,E1 254.393} C_DIS
LIN {X 0.052,Y -172.033,Z 913.385,A 0.000,B 0.000,C 90.000,E1 249.263} C_DIS
LIN {X 0.028,Y -171.462,Z 913.380,A 0.000,B 0.000,C 90.000,E1 248.411} C_DIS
LIN {X 0.008,Y -167.694,Z 913.356,A 0.000,B 0.000,C 90.000,E1 244.101} C_DIS
LIN {X 0.021,Y -166.377,Z 913.346,A 0.000,B 0.000,C 90.000,E1 242.359} C_DIS
LIN {X 0.014,Y -163.106,Z 913.327,A 0.000,B 0.000,C 90.000,E1 238.869} C_DIS
LIN {X 0.064,Y -161.053,Z 913.312,A 0.000,B 0.000,C 90.000,E1 236.215} C_DIS
LIN {X 0.047,Y -157.789,Z 913.293,A 0.000,B 0.000,C 90.000,E1 232.683} C_DIS
LIN {X -0.010,Y -155.825,Z 913.278,A 0.000,B 0.000,C 90.000,E1 230.033} C_DIS
LIN {X -0.053,Y -152.077,Z 913.253,A 0.000,B 0.000,C 90.000,E1 225.567} C_DIS
LIN {X -0.034,Y -150.327,Z 913.238,A 0.000,B 0.000,C 90.000,E1 222.852} C_DIS
LIN {X -0.012,Y -147.068,Z 913.213,A 0.000,B 0.000,C 90.000,E1 218.302} C_DIS
LIN {X 0.095,Y -145.643,Z 913.198,A 0.000,B 0.000,C 90.000,E1 215.518} C_DIS
LIN {X 0.092,Y -143.025,Z 913.172,A 0.000,B 0.000,C 90.000,E1 210.924} C_DIS
LIN {X 0.023,Y -141.651,Z 913.151,A 0.000,B 0.000,C 90.000,E1 207.257} C_DIS
LIN {X -0.057,Y -139.444,Z 913.115,A 0.000,B 0.000,C 90.000,E1 200.791} C_DIS
LIN {X -0.005,Y -139.177,Z 913.105,A 0.000,B 0.000,C 90.000,E1 198.906} C_DIS
LIN {X 0.023,Y -138.319,Z 913.053,A 0.000,B 0.000,C 90.000,E1 189.557} C_DIS
LIN {X 0.033,Y -139.468,Z 913.006,A 0.000,B 0.000,C 90.000,E1 181.146} C_DIS
LIN {X -0.026,Y -141.036,Z 912.975,A 0.000,B 0.000,C 90.000,E1 175.584} C_DIS
LIN {X 0.069,Y -142.403,Z 912.960,A 0.000,B 0.000,C 90.000,E1 172.761} C_DIS
LIN {X -0.011,Y -144.637,Z 912.934,A 0.000,B 0.000,C 90.000,E1 168.173} C_DIS
LIN {X 0.050,Y -147.832,Z 912.909,A 0.000,B 0.000,C 90.000,E1 163.559} C_DIS
LIN {X -0.005,Y -150.526,Z 912.888,A 0.000,B 0.000,C 90.000,E1 159.934} C_DIS
LIN {X 0.013,Y -153.989,Z 912.868,A 0.000,B 0.000,C 90.000,E1 156.305} C_DIS
LIN {X -0.066,Y -157.403,Z 912.848,A 0.000,B 0.000,C 90.000,E1 152.743} C_DIS
LIN {X 0.014,Y -161.609,Z 912.829,A 0.000,B 0.000,C 90.000,E1 149.154} C_DIS
LIN {X -0.021,Y -165.806,Z 912.809,A 0.000,B 0.000,C 90.000,E1 145.642} C_DIS
LIN {X 0.005,Y -170.772,Z 912.790,A 0.000,B 0.000,C 90.000,E1 142.145} C_DIS
LIN {X 0.027,Y -175.643,Z 912.771,A 0.000,B 0.000,C 90.000,E1 138.690} C_DIS
LIN {X 0.025,Y -181.258,Z 912.752,A 0.000,B 0.000,C 90.000,E1 135.283} C_DIS
LIN {X 0.026,Y -186.731,Z 912.733,A 0.000,B 0.000,C 90.000,E1 131.919} C_DIS
LIN {X -0.023,Y -191.329,Z 912.719,A 0.000,B 0.000,C 90.000,E1 129.439} C_DIS
LIN {X 0.040,Y -193.695,Z 912.711,A 0.000,B 0.000,C 90.000,E1 128.016} C_DIS
LIN {X 0.022,Y -295.346,Z 912.711,A 0.000,B 0.000,C 90.000,E1 128.016} C_DIS
LIN {X -0.100,Y -297.031,Z 912.711,A 0.000,B 0.000,C 90.000,E1 128.016} C_DIS
LIN {X -0.143,Y -301.752,Z 912.710,A 0.000,B 0.000,C 90.000,E1 127.810} C_DIS
LIN {X -0.122,Y -304.928,Z 912.708,A 0.000,B 0.000,C 90.000,E1 127.523} C_DIS
LIN {X -0.053,Y -308.600,Z 912.706,A 0.000,B 0.000,C 90.000,E1 126.996} C_DIS
LIN {X -0.029,Y -310.240,Z 912.704,A 0.000,B 0.000,C 90.000,E1 126.664} C_DIS
LIN {X 0.181,Y -311.527,Z 912.702,A 0.000,B 0.000,C 90.000,E1 126.297} C_DIS
LIN {X 0.180,Y -322.845,Z 912.682,A 0.000,B 0.000,C 90.000,E1 122.752} C_DIS
LIN {X 0.093,Y -333.453,Z 912.666,A 0.000,B 0.000,C 90.000,E1 119.922} C_DIS
LIN {X 0.103,Y -345.424,Z 912.651,A 0.000,B 0.000,C 90.000,E1 117.129} C_DIS
LIN {X 0.143,Y -358.869,Z 912.636,A 0.000,B 0.000,C 90.000,E1 114.387} C_DIS
LIN {X 0.033,Y -372.150,Z 912.622,A 0.000,B 0.000,C 90.000,E1 112.025} C_DIS
LIN {X -0.019,Y -386.782,Z 912.609,A 0.000,B 0.000,C 90.000,E1 109.704} C_DIS
LIN {X 0.173,Y -402.868,Z 912.597,A 0.000,B 0.000,C 90.000,E1 107.402} C_DIS
LIN {X 0.139,Y -420.525,Z 912.584,A 0.000,B 0.000,C 90.000,E1 105.190} C_DIS
LIN {X -0.064,Y -439.830,Z 912.573,A 0.000,B 0.000,C 90.000,E1 103.063} C_DIS
LIN {X -0.184,Y -460.018,Z 912.561,A 0.000,B 0.000,C 90.000,E1 101.074} C_DIS
LIN {X -0.182,Y -467.637,Z 912.557,A 0.000,B 0.000,C 90.000,E1 100.366} C_DIS
LIN {X -0.238,Y -469.579,Z 912.556,A 0.000,B 0.000,C 90.000,E1 100.141} C_DIS
LIN {X 0.074,Y -471.183,Z 912.555,A 0.000,B 0.000,C 90.000,E1 99.849} C_DIS
LIN {X -0.077,Y -472.387,Z 912.553,A 0.000,B 0.000,C 90.000,E1 99.613} C_DIS
LIN {X 0.028,Y -473.855,Z 912.551,A 0.000,B 0.000,C 90.000,E1 99.095} C_DIS
LIN {X 0.214,Y -474.287,Z 912.548,A 0.000,B 0.000,C 90.000,E1 98.568} C_DIS
LIN {X -0.133,Y -473.757,Z 912.545,A 0.000,B 0.000,C 90.000,E1 98.106} C_DIS
LIN {X -0.005,Y -472.186,Z 912.542,A 0.000,B 0.000,C 90.000,E1 97.587} C_DIS
LIN {X -0.146,Y -470.926,Z 912.541,A 0.000,B 0.000,C 90.000,E1 97.352} C_DIS
LIN {X 0.015,Y -450.297,Z 912.522,A 0.000,B 0.000,C 90.000,E1 94.012} C_DIS
LIN {X -0.120,Y -440.894,Z 912.514,A 0.000,B 0.000,C 90.000,E1 92.465} C_DIS
LIN {X 0.026,Y -431.267,Z 912.505,A 0.000,B 0.000,C 90.000,E1 90.859} C_DIS
LIN {X -0.197,Y -418.420,Z 912.493,A 0.000,B 0.000,C 90.000,E1 88.740} C_DIS
LIN {X 0.065,Y -407.378,Z 912.482,A 0.000,B 0.000,C 90.000,E1 86.788} C_DIS
LIN {X 0.125,Y -394.678,Z 912.470,A 0.000,B 0.000,C 90.000,E1 84.552} C_DIS
LIN {X -0.042,Y -383.643,Z 912.459,A 0.000,B 0.000,C 90.000,E1 82.591} C_DIS
LIN {X 0.045,Y -374.129,Z 912.449,A 0.000,B 0.000,C 90.000,E1 80.849} C_DIS
LIN {X -0.037,Y -364.352,Z 912.439,A 0.000,B 0.000,C 90.000,E1 79.106} C_DIS
LIN {X 0.120,Y -354.456,Z 912.430,A 0.000,B 0.000,C 90.000,E1 77.297} C_DIS
LIN {X 0.166,Y -341.145,Z 912.416,A 0.000,B 0.000,C 90.000,E1 74.866} C_DIS
LIN {X 0.093,Y -323.967,Z 912.397,A 0.000,B 0.000,C 90.000,E1 71.456} C_DIS
LIN {X -0.100,Y -313.493,Z 912.385,A 0.000,B 0.000,C 90.000,E1 69.263} C_DIS
LIN {X -0.001,Y -303.177,Z 912.372,A 0.000,B 0.000,C 90.000,E1 66.975} C_DIS
LIN {X -0.011,Y -292.884,Z 912.359,A 0.000,B 0.000,C 90.000,E1 64.665} C_DIS
LIN {X -0.098,Y -283.972,Z 912.348,A 0.000,B 0.000,C 90.000,E1 62.666} C_DIS
LIN {X -0.022,Y -273.479,Z 912.335,A 0.000,B 0.000,C 90.000,E1 60.255} C_DIS
LIN {X 0.002,Y -261.769,Z 912.319,A 0.000,B 0.000,C 90.000,E1 57.454} C_DIS
LIN {X -0.057,Y -250.718,Z 912.303,A 0.000,B 0.000,C 90.000,E1 54.609} C_DIS
LIN {X -0.093,Y -240.913,Z 912.287,A 0.000,B 0.000,C 90.000,E1 51.698} C_DIS
LIN {X 0.001,Y -230.905,Z 912.268,A 0.000,B 0.000,C 90.000,E1 48.324} C_DIS
LIN {X -0.120,Y -222.693,Z 912.252,A 0.000,B 0.000,C 90.000,E1 45.324} C_DIS
LIN {X 0.043,Y -216.872,Z 912.239,A 0.000,B 0.000,C 90.000,E1 42.975} C_DIS
LIN {X 0.057,Y -209.412,Z 912.221,A 0.000,B 0.000,C 90.000,E1 39.850} C_DIS
LIN {X -0.050,Y -202.869,Z 912.204,A 0.000,B 0.000,C 90.000,E1 36.710} C_DIS
LIN {X -0.066,Y -196.579,Z 912.186,A 0.000,B 0.000,C 90.000,E1 33.499} C_DIS
LIN {X 0.044,Y -190.827,Z 912.168,A 0.000,B 0.000,C 90.000,E1 30.207} C_DIS
LIN {X -0.016,Y -185.730,Z 912.150,A 0.000,B 0.000,C 90.000,E1 26.924} C_DIS
LIN {X 0.040,Y -181.242,Z 912.131,A 0.000,B 0.000,C 90.000,E1 23.567} C_DIS
LIN {X 0.040,Y -177.410,Z 912.112,A 0.000,B 0.000,C 90.000,E1 20.194} C_DIS
LIN {X -0.011,Y -173.658,Z 912.089,A 0.000,B 0.000,C 90.000,E1 15.953} C_DIS
LIN {X 0.043,Y -170.615,Z 912.060,A 0.000,B 0.000,C 90.000,E1 10.782} C_DIS
LIN {X 0.066,Y -168.825,Z 912.012,A 0.000,B 0.000,C 90.000,E1 2.121} C_DIS
LIN {X 0.056,Y -170.656,Z 911.969,A 0.000,B 0.000,C 90.000,E1 354.318} C_DIS
LIN {X 0.009,Y -173.681,Z 911.940,A 0.000,B 0.000,C 90.000,E1 349.162} C_DIS
LIN {X 0.063,Y -177.242,Z 911.916,A 0.000,B 0.000,C 90.000,E1 344.866} C_DIS
LIN {X -0.070,Y -180.847,Z 911.897,A 0.000,B 0.000,C 90.000,E1 341.511} C_DIS
LIN {X 0.057,Y -185.200,Z 911.878,A 0.000,B 0.000,C 90.000,E1 338.103} C_DIS
LIN {X -0.021,Y -190.451,Z 911.860,A 0.000,B 0.000,C 90.000,E1 334.793} C_DIS
LIN {X -0.070,Y -196.449,Z 911.842,A 0.000,B 0.000,C 90.000,E1 331.513} C_DIS
LIN {X -0.025,Y -202.947,Z 911.824,A 0.000,B 0.000,C 90.000,E1 328.250} C_DIS
LIN {X -0.055,Y -209.917,Z 911.806,A 0.000,B 0.000,C 90.000,E1 325.055} C_DIS
LIN {X -0.071,Y -217.409,Z 911.788,A 0.000,B 0.000,C 90.000,E1 321.904} C_DIS
LIN {X -0.013,Y -226.546,Z 911.769,A 0.000,B 0.000,C 90.000,E1 318.405} C_DIS
LIN {X -0.004,Y -235.608,Z 911.752,A 0.000,B 0.000,C 90.000,E1 315.364} C_DIS
LIN {X 0.075,Y -245.658,Z 911.735,A 0.000,B 0.000,C 90.000,E1 312.366} C_DIS
LIN {X -0.081,Y -256.881,Z 911.719,A 0.000,B 0.000,C 90.000,E1 309.483} C_DIS
LIN {X 0.131,Y -269.221,Z 911.703,A 0.000,B 0.000,C 90.000,E1 306.583} C_DIS
LIN {X -0.081,Y -284.877,Z 911.686,A 0.000,B 0.000,C 90.000,E1 303.499} C_DIS
LIN {X -0.074,Y -301.984,Z 911.669,A 0.000,B 0.000,C 90.000,E1 300.463} C_DIS
LIN {X -0.005,Y -316.435,Z 911.656,A 0.000,B 0.000,C 90.000,E1 298.153} C_DIS
LIN {X 0.058,Y -327.662,Z 911.648,A 0.000,B 0.000,C 90.000,E1 296.539} C_DIS
LIN {X 0.130,Y -344.661,Z 911.635,A 0.000,B 0.000,C 90.000,E1 294.335} C_DIS
LIN {X 0.002,Y -368.046,Z 911.620,A 0.000,B 0.000,C 90.000,E1 291.663} C_DIS
LIN {X 0.195,Y -383.941,Z 911.611,A 0.000,B 0.000,C 90.000,E1 289.939} C_DIS
LIN {X 0.016,Y -402.200,Z 911.600,A 0.000,B 0.000,C 90.000,E1 288.055} C_DIS
LIN {X -0.171,Y -414.893,Z 911.593,A 0.000,B 0.000,C 90.000,E1 286.732} C_DIS
LIN {X 0.163,Y -424.832,Z 911.587,A 0.000,B 0.000,C 90.000,E1 285.607} C_DIS
LIN {X 0.103,Y -434.446,Z 911.581,A 0.000,B 0.000,C 90.000,E1 284.537} C_DIS
LIN {X -0.181,Y -445.755,Z 911.573,A 0.000,B 0.000,C 90.000,E1 283.244} C_DIS
LIN {X -0.017,Y -454.249,Z 911.568,A 0.000,B 0.000,C 90.000,E1 282.175} C_DIS
LIN {X 0.058,Y -462.147,Z 911.562,A 0.000,B 0.000,C 90.000,E1 281.130} C_DIS
LIN {X 0.090,Y -471.413,Z 911.555,A 0.000,B 0.000,C 90.000,E1 279.849} C_DIS
LIN {X 0.046,Y -476.621,Z 911.551,A 0.000,B 0.000,C 90.000,E1 279.095} C_DIS
LIN {X 0.052,Y -481.151,Z 911.546,A 0.000,B 0.000,C 90.000,E1 278.341} C_DIS
LIN {X 0.094,Y -484.927,Z 911.542,A 0.000,B 0.000,C 90.000,E1 277.587} C_DIS
LIN {X -0.203,Y -486.992,Z 911.539,A 0.000,B 0.000,C 90.000,E1 277.125} C_DIS
LIN {X -0.002,Y -488.737,Z 911.537,A 0.000,B 0.000,C 90.000,E1 276.606} C_DIS
LIN {X 0.205,Y -490.093,Z 911.534,A 0.000,B 0.000,C 90.000,E1 276.087} C_DIS
LIN {X -0.066,Y -491.115,Z 911.531,A 0.000,B 0.000,C 90.000,E1 275.625} C_DIS
LIN {X 0.158,Y -491.808,Z 911.528,A 0.000,B 0.000,C 90.000,E1 275.106} C_DIS
LIN {X -0.103,Y -492.123,Z 911.526,A 0.000,B 0.000,C 90.000,E1 274.645} C_DIS
LIN {X 0.091,Y -492.010,Z 911.523,A 0.000,B 0.000,C 90.000,E1 274.131} C_DIS
LIN {X -0.167,Y -491.405,Z 911.520,A 0.000,B 0.000,C 90.000,E1 273.669} C_DIS
LIN {X 0.035,Y -490.348,Z 911.518,A 0.000,B 0.000,C 90.000,E1 273.154} C_DIS
LIN {X -0.230,Y -488.747,Z 911.515,A 0.000,B 0.000,C 90.000,E1 272.694} C_DIS
LIN {X -0.036,Y -486.550,Z 911.512,A 0.000,B 0.000,C 90.000,E1 272.178} C_DIS
LIN {X 0.159,Y -483.648,Z 911.509,A 0.000,B 0.000,C 90.000,E1 271.661} C_DIS
LIN {X -0.001,Y -481.943,Z 911.508,A 0.000,B 0.000,C 90.000,E1 271.432} C_DIS
LIN {X 0.153,Y -477.767,Z 911.505,A 0.000,B 0.000,C 90.000,E1 270.917} C_DIS
LIN {X -0.014,Y -475.366,Z 911.504,A 0.000,B 0.000,C 90.000,E1 270.688} C_DIS
LIN {X 0.107,Y -469.654,Z 911.501,A 0.000,B 0.000,C 90.000,E1 270.172} C_DIS
LIN {X 0.230,Y -463.692,Z 911.499,A 0.000,B 0.000,C 90.000,E1 269.714} C_DIS
LIN {X -0.188,Y -457.244,Z 911.496,A 0.000,B 0.000,C 90.000,E1 269.370} C_DIS
LIN {X -0.161,Y -450.565,Z 911.494,A 0.000,B 0.000,C 90.000,E1 269.026} C_DIS
LIN {X -0.202,Y -443.827,Z 911.493,A 0.000,B 0.000,C 90.000,E1 268.740} C_DIS
LIN {X 0.061,Y -436.671,Z 911.491,A 0.000,B 0.000,C 90.000,E1 268.453} C_DIS
LIN {X -0.207,Y -429.062,Z 911.490,A 0.000,B 0.000,C 90.000,E1 268.282} C_DIS
LIN {X -0.112,Y -420.466,Z 911.489,A 0.000,B 0.000,C 90.000,E1 268.108} C_DIS
LIN {X 0.118,Y -413.289,Z 911.489,A 0.000,B 0.000,C 90.000,E1 267.993} C_DIS
LIN {X -0.194,Y -405.109,Z 911.489,A 0.000,B 0.000,C 90.000,E1 267.993} C_DIS
LIN {X 0.069,Y -181.118,Z 911.489,A 0.000,B 0.000,C 90.000,E1 267.936} C_DIS
LIN {X -0.071,Y -180.906,Z 911.474,A 0.000,B 0.000,C 90.000,E1 265.412} C_DIS
LIN {X 0.004,Y -180.699,Z 911.470,A 0.000,B 0.000,C 90.000,E1 264.546} C_DIS
LIN {X 0.081,Y -178.784,Z 911.442,A 0.000,B 0.000,C 90.000,E1 259.454} C_DIS
LIN {X -0.017,Y -175.830,Z 911.413,A 0.000,B 0.000,C 90.000,E1 254.393} C_DIS
LIN {X -0.016,Y -172.019,Z 911.385,A 0.000,B 0.000,C 90.000,E1 249.263} C_DIS
LIN {X -0.040,Y -171.443,Z 911.380,A 0.000,B 0.000,C 90.000,E1 248.411} C_DIS
LIN {X 0.014,Y -167.678,Z 911.356,A 0.000,B 0.000,C 90.000,E1 244.076} C_DIS
LIN {X -0.046,Y -166.353,Z 911.346,A 0.000,B 0.000,C 90.000,E1 242.359} C_DIS
LIN {X -0.052,Y -163.087,Z 911.327,A 0.000,B 0.000,C 90.000,E1 238.869} C_DIS
LIN {X -0.002,Y -161.030,Z 911.312,A 0.000,B 0.000,C 90.000,E1 236.215} C_DIS
LIN {X -0.018,Y -157.770,Z 911.293,A 0.000,B 0.000,C 90.000,E1 232.683} C_DIS
LIN {X 0.045,Y -155.807,Z 911.278,A 0.000,B 0.000,C 90.000,E1 229.989} C_DIS
LIN {X -0.007,Y -152.059,Z 911.253,A 0.000,B 0.000,C 90.000,E1 225.526} C_DIS
LIN {X 0.006,Y -150.309,Z 911.238,A 0.000,B 0.000,C 90.000,E1 222.813} C_DIS
LIN {X 0.041,Y -147.053,Z 911.213,A 0.000,B 0.000,C 90.000,E1 218.257} C_DIS
LIN {X 0.033,Y -145.631,Z 911.197,A 0.000,B 0.000,C 90.000,E1 215.518} C_DIS
LIN {X 0.031,Y -143.014,Z 911.172,A 0.000,B 0.000,C 90.000,E1 210.924} C_DIS
LIN {X -0.037,Y -141.641,Z 911.151,A 0.000,B 0.000,C 90.000,E1 207.257} C_DIS
LIN {X 0.013,Y -139.439,Z 911.115,A 0.000,B 0.000,C 90.000,E1 200.737} C_DIS
LIN {X -0.065,Y -139.172,Z 911.105,A 0.000,B 0.000,C 90.000,E1 198.906} C_DIS
LIN {X -0.036,Y -138.318,Z 911.053,A 0.000,B 0.000,C 90.000,E1 189.557} C_DIS
LIN {X -0.027,Y -139.472,Z 911.006,A 0.000,B 0.000,C 90.000,E1 181.146} C_DIS
LIN {X 0.053,Y -141.046,Z 910.975,A 0.000,B 0.000,C 90.000,E1 175.527} C_DIS
LIN {X 0.008,Y -142.416,Z 910.960,A 0.000,B 0.000,C 90.000,E1 172.761} C_DIS
LIN {X -0.072,Y -144.650,Z 910.934,A 0.000,B 0.000,C 90.000,E1 168.173} C_DIS
LIN {X -0.013,Y -147.847,Z 910.909,A 0.000,B 0.000,C 90.000,E1 163.559} C_DIS
LIN {X 0.073,Y -150.546,Z 910.888,A 0.000,B 0.000,C 90.000,E1 159.880} C_DIS
LIN {X -0.050,Y -154.013,Z 910.868,A 0.000,B 0.000,C 90.000,E1 156.305} C_DIS
LIN {X 0.009,Y -157.427,Z 910.848,A 0.000,B 0.000,C 90.000,E1 152.692} C_DIS
LIN {X 0.030,Y -161.640,Z 910.829,A 0.000,B 0.000,C 90.000,E1 149.125} C_DIS
LIN {X 0.049,Y -165.836,Z 910.809,A 0.000,B 0.000,C 90.000,E1 145.595} C_DIS
LIN {X 0.041,Y -170.808,Z 910.790,A 0.000,B 0.000,C 90.000,E1 142.110} C_DIS
LIN {X -0.042,Y -175.677,Z 910.770,A 0.000,B 0.000,C 90.000,E1 138.690} C_DIS
LIN {X 0.081,Y -181.291,Z 910.751,A 0.000,B 0.000,C 90.000,E1 135.243} C_DIS
LIN {X -0.046,Y -186.770,Z 910.733,A 0.000,B 0.000,C 90.000,E1 131.919} C_DIS
LIN {X 0.026,Y -191.364,Z 910.719,A 0.000,B 0.000,C 90.000,E1 129.402} C_DIS
LIN {X 0.008,Y -193.650,Z 910.711,A 0.000,B 0.000,C 90.000,E1 128.051} C_DIS
LIN {X 0.141,Y -294.807,Z 910.711,A 0.000,B 0.000,C 90.000,E1 128.016} C_DIS
LIN {X 0.062,Y -300.069,Z 910.711,A 0.000,B 0.000,C 90.000,E1 127.890} C_DIS
LIN {X 0.166,Y -302.261,Z 910.710,A 0.000,B 0.000,C 90.000,E1 127.729} C_DIS
LIN {X 0.041,Y -306.120,Z 910.708,A 0.000,B 0.000,C 90.000,E1 127.363} C_DIS
LIN {X 0.056,Y -309.602,Z 910.704,A 0.000,B 0.000,C 90.000,E1 126.790} C_DIS
LIN {X 0.084,Y -311.005,Z 910.703,A 0.000,B 0.000,C 90.000,E1 126.457} C_DIS
LIN {X -0.116,Y -314.034,Z 910.697,A 0.000,B 0.000,C 90.000,E1 125.518} C_DIS
LIN {X -0.035,Y -324.578,Z 910.679,A 0.000,B 0.000,C 90.000,E1 122.291} C_DIS
LIN {X -0.074,Y -335.415,Z 910.664,A 0.000,B 0.000,C 90.000,E1 119.461} C_DIS
LIN {X -0.018,Y -347.638,Z 910.648,A 0.000,B 0.000,C 90.000,E1 116.668} C_DIS
LIN {X -0.071,Y -361.346,Z 910.633,A 0.000,B 0.000,C 90.000,E1 113.951} C_DIS
LIN {X -0.127,Y -374.884,Z 910.620,A 0.000,B 0.000,C 90.000,E1 111.589} C_DIS
LIN {X -0.118,Y -389.791,Z 910.607,A 0.000,B 0.000,C 90.000,E1 109.268} C_DIS
LIN {X 0.018,Y -406.176,Z 910.594,A 0.000,B 0.000,C 90.000,E1 106.985} C_DIS
LIN {X 0.059,Y -424.154,Z 910.582,A 0.000,B 0.000,C 90.000,E1 104.773} C_DIS
LIN {X 0.013,Y -443.713,Z 910.570,A 0.000,B 0.000,C 90.000,E1 102.647} C_DIS
LIN {X 0.159,Y -464.011,Z 910.559,A 0.000,B 0.000,C 90.000,E1 100.658} C_DIS
LIN {X 0.074,Y -466.599,Z 910.558,A 0.000,B 0.000,C 90.000,E1 100.433} C_DIS
LIN {X 0.104,Y -468.800,Z 910.557,A 0.000,B 0.000,C 90.000,E1 100.197} C_DIS
LIN {X 0.132,Y -470.463,Z 910.555,A 0.000,B 0.000,C 90.000,E1 99.962} C_DIS
LIN {X -0.016,Y -471.845,Z 910.554,A 0.000,B 0.000,C 90.000,E1 99.726} C_DIS
LIN {X -0.244,Y -472.872,Z 910.553,A 0.000,B 0.000,C 90.000,E1 99.500} C_DIS
LIN {X -0.060,Y -474.055,Z 910.550,A 0.000,B 0.000,C 90.000,E1 98.973} C_DIS
LIN {X 0.056,Y -474.238,Z 910.547,A 0.000,B 0.000,C 90.000,E1 98.454} C_DIS
LIN {X 0.181,Y -473.453,Z 910.544,A 0.000,B 0.000,C 90.000,E1 97.936} C_DIS
LIN {X -0.097,Y -471.575,Z 910.541,A 0.000,B 0.000,C 90.000,E1 97.466} C_DIS
LIN {X 0.023,Y -468.436,Z 910.539,A 0.000,B 0.000,C 90.000,E1 96.947} C_DIS
LIN {X -0.155,Y -449.521,Z 910.522,A 0.000,B 0.000,C 90.000,E1 93.898} C_DIS
LIN {X 0.141,Y -440.135,Z 910.513,A 0.000,B 0.000,C 90.000,E1 92.293} C_DIS
LIN {X -0.162,Y -430.488,Z 910.504,A 0.000,B 0.000,C 90.000,E1 90.745} C_DIS
LIN {X -0.091,Y -419.242,Z 910.494,A 0.000,B 0.000,C 90.000,E1 88.854} C_DIS
LIN {X -0.147,Y -406.590,Z 910.481,A 0.000,B 0.000,C 90.000,E1 86.674} C_DIS
LIN {X -0.127,Y -395.460,Z 910.471,A 0.000,B 0.000,C 90.000,E1 84.723} C_DIS
LIN {X 0.111,Y -384.423,Z 910.460,A 0.000,B 0.000,C 90.000,E1 82.704} C_DIS
LIN {X 0.164,Y -373.318,Z 910.448,A 0.000,B 0.000,C 90.000,E1 80.679} C_DIS
LIN {X 0.128,Y -363.510,Z 910.439,A 0.000,B 0.000,C 90.000,E1 78.926} C_DIS
LIN {X -0.076,Y -353.656,Z 910.429,A 0.000,B 0.000,C 90.000,E1 77.173} C_DIS
LIN {X -0.124,Y -340.371,Z 910.415,A 0.000,B 0.000,C 90.000,E1 74.755} C_DIS
LIN {X -0.114,Y -323.255,Z 910.396,A 0.000,B 0.000,C 90.000,E1 71.329} C_DIS
LIN {X -0.020,Y -312.793,Z 910.384,A 0.000,B 0.000,C 90.000,E1 69.082} C_DIS
LIN {X 0.059,Y -302.495,Z 910.371,A 0.000,B 0.000,C 90.000,E1 66.794} C_DIS
LIN {X 0.017,Y -290.767,Z 910.356,A 0.000,B 0.000,C 90.000,E1 64.152} C_DIS
LIN {X -0.108,Y -281.817,Z 910.345,A 0.000,B 0.000,C 90.000,E1 62.153} C_DIS
LIN {X -0.144,Y -269.866,Z 910.330,A 0.000,B 0.000,C 90.000,E1 59.410} C_DIS
LIN {X -0.071,Y -258.322,Z 910.314,A 0.000,B 0.000,C 90.000,E1 56.580} C_DIS
LIN {X -0.084,Y -248.919,Z 910.300,A 0.000,B 0.000,C 90.000,E1 54.069} C_DIS
LIN {X 0.111,Y -238.233,Z 910.282,A 0.000,B 0.000,C 90.000,E1 50.723} C_DIS
LIN {X -0.040,Y -228.475,Z 910.263,A 0.000,B 0.000,C 90.000,E1 47.391} C_DIS
LIN {X -0.064,Y -220.485,Z 910.246,A 0.000,B 0.000,C 90.000,E1 44.352} C_DIS
LIN {X 0.034,Y -212.791,Z 910.229,A 0.000,B 0.000,C 90.000,E1 41.229} C_DIS
LIN {X -0.019,Y -205.874,Z 910.212,A 0.000,B 0.000,C 90.000,E1 38.096} C_DIS
LIN {X -0.005,Y -199.534,Z 910.194,A 0.000,B 0.000,C 90.000,E1 34.898} C_DIS
